C01819=1221.281,-16.840,-40.871,-179.722,5.391,148.856
C01820=1221.286,-17.090,-40.856,-179.724,5.391,148.857
C01821=1221.291,-17.339,-40.844,-179.727,5.391,148.857
C01822=1221.296,-17.589,-40.830,-179.729,5.390,148.858
C01823=1221.302,-17.838,-40.816,-179.732,5.390,148.859
C01824=1221.306,-18.088,-40.803,-179.734,5.390,148.859
C01825=1221.312,-18.337,-40.789,-179.737,5.390,148.860
C01826=1221.316,-18.587,-40.776,-179.739,5.389,148.861
C01827=1221.321,-18.837,-40.762,-179.741,5.389,148.861
C01828=1221.327,-19.086,-40.748,-179.744,5.389,148.862
C01829=1221.331,-19.336,-40.735,-179.747,5.388,148.863
C01830=1221.337,-19.585,-40.721,-179.749,5.389,148.863
C01831=1221.342,-19.835,-40.707,-179.752,5.388,148.864
C01832=1221.347,-20.084,-40.695,-179.754,5.388,148.865
C01833=1221.352,-20.334,-40.680,-179.756,5.388,148.866
C01834=1221.357,-20.583,-40.668,-179.759,5.388,148.866
C01835=1221.362,-20.833,-40.653,-179.762,5.387,148.867
C01836=1221.367,-21.082,-40.641,-179.764,5.387,148.868
C01837=1221.373,-21.333,-40.627,-179.766,5.387,148.868
C01838=1221.378,-21.582,-40.613,-179.769,5.386,148.869
C01839=1221.383,-21.832,-40.600,-179.772,5.386,148.870
C01840=1221.388,-22.081,-40.586,-179.774,5.386,148.870
C01841=1221.393,-22.350,-40.573,-179.776,5.386,148.871
C01842=1221.399,-22.620,-40.558,-179.779,5.385,148.872
C01843=1221.404,-22.889,-40.543,-179.782,5.385,148.873
C01844=1221.410,-23.158,-40.530,-179.784,5.384,148.873
C01845=1221.415,-23.408,-40.515,-179.786,5.384,148.874
C01846=1221.420,-23.657,-40.503,-179.789,5.384,148.875
C01847=1221.425,-23.908,-40.489,-179.792,5.383,148.875
C01848=1221.430,-24.156,-40.476,-179.794,5.384,148.876
C01849=1221.435,-24.407,-40.462,-179.797,5.383,148.877
C01850=1221.440,-24.656,-40.450,-179.799,5.383,148.877
C01851=1221.445,-24.906,-40.435,-179.801,5.383,148.878
C01852=1221.450,-25.155,-40.423,-179.804,5.383,148.879
C01853=1221.456,-25.405,-40.409,-179.807,5.382,148.879
C01854=1221.461,-25.654,-40.396,-179.809,5.382,148.880
C01855=1221.466,-25.904,-40.382,-179.811,5.382,148.881
C01856=1221.471,-26.154,-40.370,-179.814,5.381,148.882
C01857=1221.476,-26.403,-40.355,-179.816,5.382,148.882
C01858=1221.481,-26.653,-40.343,-179.819,5.381,148.883
C01859=1221.486,-26.903,-40.329,-179.821,5.381,148.884
C01860=1221.491,-27.152,-40.316,-179.823,5.381,148.884
C01861=1221.496,-27.401,-40.303,-179.826,5.381,148.885
C01862=1221.501,-27.651,-40.290,-179.829,5.380,148.886
C01863=1221.507,-27.901,-40.277,-179.831,5.380,148.886
C01864=1221.512,-28.150,-40.263,-179.834,5.380,148.887
C01865=1221.517,-28.400,-40.250,-179.836,5.379,148.888
C01866=1221.521,-28.650,-40.237,-179.838,5.380,148.889
C01867=1221.527,-28.899,-40.224,-179.841,5.379,148.889
C01868=1221.532,-29.149,-40.211,-179.844,5.379,148.890
C01869=1221.537,-29.398,-40.197,-179.846,5.379,148.891
C01870=1221.542,-29.648,-40.185,-179.848,5.379,148.891
C01871=1221.547,-29.898,-40.172,-179.851,5.378,148.892
C01872=1221.553,-30.147,-40.158,-179.853,5.378,148.893
C01873=1221.557,-30.397,-40.146,-179.856,5.378,148.893
C01874=1221.562,-30.646,-40.132,-179.858,5.377,148.894
C01875=1221.568,-30.896,-40.119,-179.860,5.378,148.895
C01876=1221.572,-31.146,-40.106,-179.863,5.377,148.896
C01877=1221.578,-31.395,-40.093,-179.866,5.377,148.896
C01878=1221.583,-31.645,-40.080,-179.868,5.377,148.897
C01879=1221.588,-31.895,-40.067,-179.871,5.377,148.898
C01880=1221.594,-32.144,-40.054,-179.873,5.376,148.898
C01881=1221.598,-32.394,-40.041,-179.875,5.376,148.899
C01882=1221.603,-32.643,-40.028,-179.878,5.376,148.900
C01883=1221.608,-32.892,-40.015,-179.881,5.375,148.900
C01884=1221.613,-33.143,-40.002,-179.883,5.376,148.901
C01885=1221.619,-33.392,-39.989,-179.885,5.375,148.902
C01886=1221.624,-33.641,-39.976,-179.888,5.375,148.903
C01887=1221.629,-33.892,-39.963,-179.890,5.375,148.903
C01888=1221.634,-34.141,-39.950,-179.893,5.375,148.904
C01889=1221.639,-34.390,-39.938,-179.895,5.375,148.905
C01890=1221.644,-34.641,-39.924,-179.897,5.374,148.905
C01891=1221.650,-34.890,-39.912,-179.900,5.374,148.906
C01892=1221.655,-35.139,-39.899,-179.902,5.374,148.907
C01893=1221.659,-35.389,-39.886,-179.905,5.374,148.907
C01894=1221.665,-35.639,-39.873,-179.908,5.373,148.908
C01895=1221.670,-35.888,-39.860,-179.910,5.374,148.909
C01896=1221.675,-36.138,-39.847,-179.912,5.373,148.910
C01897=1221.680,-36.388,-39.835,-179.915,5.373,148.910
C01898=1221.686,-36.637,-39.821,-179.917,5.373,148.911
C01899=1221.690,-36.887,-39.808,-179.920,5.373,148.912
C01900=1221.695,-37.137,-39.796,-179.922,5.372,148.912
C01901=1221.700,-37.386,-39.783,-179.924,5.372,148.913
C01902=1221.705,-37.636,-39.770,-179.927,5.372,148.913
C01903=1221.711,-37.886,-39.757,-179.929,5.372,148.914
C01904=1221.716,-38.135,-39.744,-179.931,5.371,148.915
C01905=1221.721,-38.384,-39.732,-179.934,5.371,148.916
C01906=1221.726,-38.634,-39.719,-179.936,5.371,148.916
C01907=1221.731,-38.883,-39.706,-179.939,5.371,148.917
C01908=1221.737,-39.133,-39.693,-179.941,5.370,148.918
C01909=1221.741,-39.383,-39.680,-179.944,5.371,148.918
C01910=1221.746,-39.632,-39.668,-179.946,5.370,148.919
C01911=1221.752,-39.882,-39.656,-179.949,5.370,148.920
C01912=1221.757,-40.132,-39.643,-179.951,5.370,148.920
C01913=1221.761,-40.382,-39.630,-179.954,5.369,148.921
C01914=1221.767,-40.631,-39.617,-179.956,5.370,148.922
C01915=1221.772,-40.881,-39.604,-179.958,5.369,148.923
C01916=1221.777,-41.130,-39.592,-179.961,5.369,148.923
C01917=1221.782,-41.380,-39.579,-179.963,5.369,148.924
C01918=1221.787,-41.630,-39.567,-179.966,5.369,148.925
C01919=1221.793,-41.879,-39.554,-179.968,5.368,148.925
C01920=1221.798,-42.129,-39.542,-179.971,5.368,148.926
C01921=1221.803,-42.379,-39.528,-179.973,5.368,148.927
C01922=1221.808,-42.628,-39.515,-179.975,5.368,148.927
C01923=1221.813,-42.878,-39.503,-179.978,5.368,148.928
C01924=1221.819,-43.127,-39.491,-179.981,5.367,148.929
C01925=1221.823,-43.378,-39.478,-179.983,5.368,148.930
C01926=1221.828,-43.627,-39.465,-179.985,5.367,148.930
C01927=1221.833,-43.876,-39.453,-179.988,5.367,148.931
C01928=1221.839,-44.125,-39.440,-179.990,5.367,148.932
C01929=1221.844,-44.375,-39.428,-179.993,5.367,148.932
C01930=1221.848,-44.625,-39.415,-179.995,5.367,148.933
C01931=1221.854,-44.875,-39.403,-179.998,5.366,148.934
C01932=1221.859,-45.124,-39.390,180.000,5.366,148.935
C01933=1221.864,-45.374,-39.378,179.998,5.366,148.935
C01934=1221.870,-45.624,-39.365,179.995,5.366,148.936
C01935=1221.875,-45.874,-39.352,179.993,5.366,148.937
C01936=1221.880,-46.124,-39.340,179.990,5.366,148.937
C01937=1221.885,-46.373,-39.328,179.988,5.365,148.938
C01938=1221.890,-46.622,-39.315,179.986,5.366,148.939
C01939=1221.896,-46.872,-39.303,179.983,5.365,148.939
C01940=1221.901,-47.121,-39.291,179.981,5.365,148.940
C01941=1221.905,-47.371,-39.278,179.978,5.365,148.941
C01942=1221.911,-47.621,-39.266,179.975,5.364,148.942
C01943=1221.916,-47.871,-39.253,179.973,5.365,148.942
C01944=1221.921,-48.120,-39.240,179.971,5.364,148.943
C01945=1221.926,-48.390,-39.228,179.968,5.364,148.944
C01946=1221.932,-48.659,-39.214,179.966,5.364,148.944
C01947=1221.938,-48.930,-39.201,179.963,5.364,148.945
C01948=1221.943,-49.200,-39.187,179.960,5.364,148.946
C01949=1221.948,-49.449,-39.174,179.958,5.364,148.947
C01950=1221.953,-49.699,-39.162,179.956,5.363,148.947
C01951=1221.959,-49.948,-39.150,179.953,5.363,148.948
C01952=1221.964,-50.198,-39.138,179.951,5.363,148.949
C01953=1221.969,-50.448,-39.125,179.948,5.362,148.949
C01954=1221.974,-50.697,-39.113,179.946,5.363,148.950
C01955=1221.978,-50.947,-39.101,179.944,5.362,148.951
C01956=1221.983,-51.197,-39.089,179.941,5.362,148.951
C01957=1221.989,-51.447,-39.077,179.939,5.362,148.952
C01958=1221.994,-51.696,-39.064,179.936,5.362,148.953
C01959=1221.999,-51.946,-39.052,179.934,5.362,148.953
C01960=1222.005,-52.195,-39.040,179.932,5.362,148.954
C01961=1222.010,-52.445,-39.028,179.929,5.361,148.955
C01962=1222.015,-52.694,-39.015,179.927,5.361,148.956
C01963=1222.021,-52.944,-39.003,179.924,5.361,148.956
C01964=1222.026,-53.194,-38.991,179.922,5.361,148.957
C01965=1222.030,-53.444,-38.979,179.919,5.361,148.958
C01966=1222.035,-53.693,-38.966,179.917,5.360,148.958
C01967=1222.040,-53.943,-38.954,179.915,5.361,148.959
C01968=1222.045,-54.193,-38.942,179.912,5.360,148.960
C01969=1222.051,-54.442,-38.930,179.910,5.361,148.961
C01970=1222.056,-54.692,-38.917,179.907,5.360,148.961
C01971=1222.061,-54.942,-38.905,179.905,5.360,148.962
C01972=1222.066,-55.191,-38.893,179.902,5.360,148.963
C01973=1222.071,-55.441,-38.882,179.900,5.359,148.963
C01974=1222.076,-55.690,-38.869,179.898,5.360,148.964
C01975=1222.082,-55.940,-38.857,179.895,5.359,148.965
C01976=1222.087,-56.190,-38.845,179.893,5.360,148.965
C01977=1222.092,-56.439,-38.833,179.890,5.359,148.966
C01978=1222.097,-56.689,-38.821,179.888,5.359,148.967
C01979=1222.102,-56.938,-38.809,179.886,5.359,148.968
C01980=1222.108,-57.188,-38.797,179.883,5.359,148.968
C01981=1222.113,-57.438,-38.785,179.881,5.359,148.969
C01982=1222.117,-57.687,-38.773,179.878,5.358,148.970
C01983=1222.122,-57.938,-38.761,179.876,5.359,148.970
C01984=1222.127,-58.187,-38.748,179.873,5.358,148.971
C01985=1222.133,-58.437,-38.736,179.871,5.358,148.972
C01986=1222.138,-58.687,-38.724,179.869,5.358,148.972
C01987=1222.143,-58.936,-38.712,179.866,5.358,148.973
C01988=1222.148,-59.186,-38.700,179.864,5.358,148.974
C01989=1222.153,-59.436,-38.689,179.862,5.357,148.974
C01990=1222.159,-59.685,-38.676,179.859,5.357,148.975
C01991=1222.163,-59.935,-38.665,179.857,5.357,148.976
C01992=1222.169,-60.185,-38.653,179.854,5.357,148.976
C01993=1222.174,-60.435,-38.641,179.852,5.357,148.977
C01994=1222.179,-60.684,-38.628,179.850,5.356,148.978
C01995=1222.184,-60.933,-38.617,179.847,5.357,148.979
C01996=1222.190,-61.183,-38.605,179.845,5.356,148.979
C01997=1222.195,-61.432,-38.593,179.842,5.356,148.980
C01998=1222.200,-61.682,-38.582,179.840,5.356,148.981
C01999=1222.205,-61.932,-38.570,179.837,5.356,148.981
C02000=1222.211,-62.181,-38.558,179.835,5.356,148.982
C02001=1222.215,-62.430,-38.546,179.833,5.356,148.983
C02002=1222.220,-62.680,-38.534,179.831,5.356,148.984
C02003=1222.226,-62.930,-38.522,179.828,5.356,148.984
C02004=1222.231,-63.180,-38.510,179.825,5.355,148.985
C02005=1222.236,-63.430,-38.499,179.823,5.355,148.986
C02006=1222.241,-63.679,-38.486,179.820,5.355,148.986
C02007=1222.247,-63.929,-38.474,179.818,5.355,148.987
C02008=1222.251,-64.179,-38.463,179.816,5.355,148.988
C02009=1222.257,-64.429,-38.451,179.814,5.355,148.988
C02010=1222.261,-64.678,-38.440,179.811,5.355,148.989
C02011=1222.267,-64.928,-38.427,179.809,5.355,148.990
C02012=1222.272,-65.178,-38.415,179.806,5.355,148.991
C02013=1222.277,-65.427,-38.404,179.803,5.354,148.991
C02014=1222.283,-65.676,-38.393,179.801,5.354,148.992
C02015=1222.288,-65.926,-38.381,179.799,5.354,148.993
C02016=1222.293,-66.176,-38.369,179.797,5.354,148.993
C02017=1222.298,-66.426,-38.358,179.794,5.354,148.994
C02018=1222.303,-66.675,-38.345,179.792,5.354,148.995
C02019=1222.308,-66.925,-38.334,179.790,5.353,148.995
C02020=1222.313,-67.175,-38.322,179.788,5.354,148.996
C02021=1222.318,-67.425,-38.310,179.785,5.353,148.997
C02022=1222.324,-67.674,-38.299,179.782,5.353,148.997
C02023=1222.329,-67.924,-38.287,179.780,5.353,148.998
C02024=1222.334,-68.173,-38.276,179.778,5.353,148.999
C02025=1222.340,-68.423,-38.264,179.775,5.353,149.000
C02026=1222.344,-68.673,-38.253,179.773,5.353,149.000
C02027=1222.350,-68.923,-38.241,179.771,5.353,149.001
C02028=1222.355,-69.172,-38.229,179.768,5.352,149.002
C02029=1222.360,-69.422,-38.218,179.766,5.353,149.002
C02030=1222.365,-69.672,-38.206,179.763,5.352,149.003
C02031=1222.371,-69.921,-38.195,179.761,5.352,149.004
C02032=1222.376,-70.171,-38.183,179.758,5.352,149.005
C02033=1222.381,-70.421,-38.172,179.756,5.352,149.005
C02034=1222.386,-70.671,-38.160,179.754,5.352,149.006
C02035=1222.391,-70.920,-38.148,179.751,5.352,149.007
C02036=1222.396,-71.170,-38.136,179.749,5.352,149.007
C02037=1222.401,-71.420,-38.125,179.746,5.352,149.008
C02038=1222.407,-71.669,-38.114,179.744,5.352,149.009
C02039=1222.412,-71.919,-38.102,179.742,5.351,149.009
C02040=1222.417,-72.169,-38.091,179.739,5.352,149.010
C02041=1222.422,-72.418,-38.079,179.737,5.351,149.011
C02042=1222.427,-72.668,-38.067,179.735,5.351,149.011
C02043=1222.433,-72.917,-38.056,179.733,5.351,149.012
C02044=1222.438,-73.167,-38.045,179.730,5.350,149.013
C02045=1222.443,-73.417,-38.033,179.728,5.351,149.013
C02046=1222.448,-73.667,-38.021,179.725,5.350,149.014
C02047=1222.453,-73.916,-38.010,179.723,5.351,149.015
C02048=1222.459,-74.166,-37.999,179.720,5.350,149.016
C02049=1222.465,-74.437,-37.986,179.718,5.351,149.016
C02050=1222.469,-74.707,-37.974,179.715,5.350,149.017
C02051=1222.475,-74.977,-37.962,179.712,5.350,149.018
C02052=1222.481,-75.248,-37.950,179.710,5.350,149.019
C02053=1222.486,-75.498,-37.938,179.708,5.350,149.019
C02054=1222.492,-75.747,-37.927,179.706,5.350,149.020
C02055=1222.496,-75.996,-37.916,179.703,5.350,149.021
C02056=1222.502,-76.246,-37.904,179.700,5.349,149.022
C02057=1222.506,-76.496,-37.893,179.698,5.350,149.022
C02058=1222.512,-76.746,-37.881,179.695,5.349,149.023
C02059=1222.518,-76.995,-37.870,179.693,5.350,149.024
C02060=1222.523,-77.245,-37.859,179.691,5.349,149.024
C02061=1222.528,-77.495,-37.847,179.689,5.349,149.025
C02062=1222.532,-77.745,-37.836,179.686,5.349,149.026
C02063=1222.538,-77.994,-37.824,179.684,5.349,149.026
C02064=1222.543,-78.244,-37.814,179.682,5.349,149.027
C02065=1222.548,-78.494,-37.803,179.680,5.349,149.028
C02066=1222.553,-78.744,-37.791,179.677,5.349,149.028
C02067=1222.559,-78.993,-37.780,179.675,5.349,149.029
C02068=1222.564,-79.243,-37.769,179.672,5.348,149.030
C02069=1222.569,-79.493,-37.757,179.670,5.349,149.030
C02070=1222.574,-79.742,-37.746,179.667,5.348,149.031
C02071=1222.580,-79.992,-37.734,179.665,5.348,149.032
C02072=1222.585,-80.242,-37.724,179.663,5.348,149.033
C02073=1222.590,-80.491,-37.713,179.660,5.348,149.033
C02074=1222.596,-80.741,-37.701,179.658,5.348,149.034
C02075=1222.600,-80.990,-37.690,179.655,5.348,149.035
C02076=1222.605,-81.241,-37.679,179.654,5.348,149.035
C02077=1222.611,-81.490,-37.668,179.651,5.347,149.036
C02078=1222.616,-81.739,-37.656,179.649,5.348,149.037
C02079=1222.621,-81.990,-37.646,179.646,5.347,149.037
C02080=1222.626,-82.239,-37.635,179.644,5.347,149.038
C02081=1222.632,-82.488,-37.623,179.641,5.347,149.039
C02082=1222.637,-82.739,-37.612,179.639,5.347,149.039
C02083=1222.641,-82.988,-37.601,179.637,5.347,149.040
C02084=1222.647,-83.238,-37.590,179.635,5.347,149.041
C02085=1222.652,-83.488,-37.579,179.632,5.347,149.042
C02086=1222.657,-83.737,-37.568,179.630,5.347,149.042
C02087=1222.662,-83.986,-37.557,179.627,5.347,149.043
C02088=1222.668,-84.237,-37.546,179.625,5.347,149.044
C02089=1222.673,-84.487,-37.534,179.622,5.347,149.044
C02090=1222.678,-84.735,-37.523,179.620,5.347,149.045
C02091=1222.683,-84.986,-37.513,179.618,5.346,149.046
C02092=1222.689,-85.236,-37.501,179.616,5.347,149.046
C02093=1222.694,-85.485,-37.491,179.613,5.346,149.047
C02094=1222.699,-85.735,-37.480,179.611,5.346,149.048
C02095=1222.704,-85.984,-37.468,179.609,5.346,149.048
C02096=1222.709,-86.234,-37.458,179.606,5.346,149.049
C02097=1222.715,-86.484,-37.446,179.604,5.346,149.050
C02098=1222.720,-86.733,-37.436,179.602,5.346,149.051
C02099=1222.725,-86.983,-37.425,179.599,5.346,149.051
C02100=1222.730,-87.233,-37.414,179.596,5.345,149.052
C02101=1222.735,-87.482,-37.403,179.594,5.346,149.053
C02102=1222.741,-87.733,-37.392,179.592,5.345,149.053
C02103=1222.746,-87.982,-37.381,179.589,5.346,149.054
C02104=1222.751,-88.232,-37.370,179.587,5.345,149.055
C02105=1222.756,-88.482,-37.359,179.585,5.345,149.055
C02106=1222.762,-88.731,-37.349,179.583,5.345,149.056
C02107=1222.766,-88.981,-37.338,179.580,5.345,149.057
C02108=1222.772,-89.231,-37.327,179.578,5.345,149.058
C02109=1222.777,-89.480,-37.316,179.576,5.345,149.058
C02110=1222.782,-89.731,-37.305,179.573,5.345,149.059
C02111=1222.788,-89.979,-37.294,179.571,5.345,149.060
C02112=1222.793,-90.230,-37.284,179.568,5.345,149.060
C02113=1222.797,-90.479,-37.272,179.566,5.345,149.061
C02114=1222.803,-90.729,-37.262,179.563,5.344,149.062
C02115=1222.808,-90.979,-37.250,179.561,5.345,149.062
C02116=1222.814,-91.228,-37.240,179.559,5.344,149.063
C02117=1222.819,-91.478,-37.229,179.557,5.344,149.064
C02118=1222.824,-91.728,-37.218,179.554,5.344,149.064
C02119=1222.829,-91.978,-37.208,179.552,5.344,149.065
C02120=1222.834,-92.227,-37.197,179.550,5.344,149.066
C02121=1222.839,-92.477,-37.186,179.548,5.344,149.067
C02122=1222.844,-92.727,-37.175,179.545,5.344,149.067
C02123=1222.850,-92.976,-37.165,179.543,5.344,149.068
C02124=1222.855,-93.226,-37.154,179.540,5.344,149.069
C02125=1222.860,-93.475,-37.143,179.538,5.344,149.069
C02126=1222.866,-93.726,-37.132,179.536,5.343,149.070
C02127=1222.871,-93.975,-37.122,179.534,5.344,149.071
C02128=1222.876,-94.225,-37.111,179.531,5.343,149.071
C02129=1222.882,-94.475,-37.100,179.529,5.343,149.072
C02130=1222.887,-94.725,-37.090,179.526,5.343,149.073
C02131=1222.892,-94.974,-37.079,179.524,5.343,149.073
C02132=1222.897,-95.224,-37.068,179.522,5.343,149.074
C02133=1222.903,-95.473,-37.058,179.519,5.343,149.075
C02134=1222.907,-95.723,-37.047,179.517,5.343,149.076
C02135=1222.913,-95.973,-37.037,179.515,5.343,149.076
C02136=1222.918,-96.223,-37.026,179.512,5.343,149.077
C02137=1222.923,-96.472,-37.015,179.510,5.343,149.077
C02138=1222.928,-96.722,-37.005,179.508,5.342,149.078
C02139=1222.934,-96.972,-36.994,179.506,5.343,149.079
C02140=1222.939,-97.222,-36.984,179.503,5.342,149.080
C02141=1222.944,-97.471,-36.973,179.501,5.343,149.080
C02142=1222.949,-97.721,-36.962,179.498,5.342,149.081
C02143=1222.955,-97.971,-36.952,179.496,5.343,149.082
C02144=1222.960,-98.221,-36.942,179.494,5.343,149.082
C02145=1222.965,-98.470,-36.931,179.491,5.343,149.083
C02146=1222.970,-98.720,-36.920,179.490,5.343,149.084
C02147=1222.975,-98.970,-36.910,179.487,5.342,149.084
C02148=1222.980,-99.220,-36.899,179.485,5.342,149.085
C02149=1222.986,-99.469,-36.888,179.482,5.342,149.086
C02150=1222.991,-99.719,-36.878,179.480,5.342,149.086
C02151=1222.996,-99.968,-36.868,179.478,5.342,149.087
C02152=1223.001,-100.219,-36.857,179.475,5.342,149.088
C02153=1223.007,-100.489,-36.846,179.473,5.342,149.089
C02154=1223.013,-100.760,-36.834,179.470,5.341,149.089
C02155=1223.018,-101.032,-36.823,179.468,5.342,149.090
C02156=1223.024,-101.303,-36.812,179.465,5.341,149.091
C02157=1223.029,-101.553,-36.801,179.463,5.342,149.091
C02158=1223.035,-101.802,-36.791,179.461,5.341,149.092
C02159=1223.039,-102.052,-36.781,179.459,5.342,149.093
C02160=1223.045,-102.301,-36.770,179.456,5.341,149.094
C02161=1223.050,-102.551,-36.760,179.454,5.342,149.094
C02162=1223.055,-102.801,-36.750,179.451,5.341,149.095
C02163=1223.061,-103.050,-36.739,179.449,5.341,149.096
C02164=1223.066,-103.301,-36.729,179.447,5.341,149.096
C02165=1223.071,-103.550,-36.719,179.445,5.341,149.097
C02166=1223.076,-103.800,-36.707,179.442,5.341,149.098
C02167=1223.081,-104.049,-36.698,179.440,5.341,149.098
C02168=1223.087,-104.299,-36.687,179.437,5.341,149.099
C02169=1223.092,-104.549,-36.677,179.435,5.341,149.100
C02170=1223.097,-104.798,-36.667,179.432,5.341,149.101
C02171=1223.102,-105.049,-36.656,179.431,5.341,149.101
C02172=1223.108,-105.298,-36.646,179.428,5.340,149.102
C02173=1223.113,-105.548,-36.636,179.426,5.341,149.102
C02174=1223.118,-105.798,-36.626,179.424,5.341,149.103
C02175=1223.123,-106.047,-36.616,179.421,5.340,149.104
C02176=1223.129,-106.297,-36.605,179.419,5.341,149.105
C02177=1223.134,-106.547,-36.595,179.417,5.340,149.105
C02178=1223.139,-106.797,-36.585,179.414,5.341,149.106
C02179=1223.144,-107.047,-36.575,179.412,5.340,149.107
C02180=1223.149,-107.296,-36.564,179.410,5.340,149.107
C02181=1223.155,-107.546,-36.554,179.408,5.340,149.108
C02182=1223.160,-107.796,-36.544,179.405,5.340,149.109
C02183=1223.165,-108.045,-36.533,179.403,5.340,149.109
C02184=1223.170,-108.295,-36.524,179.401,5.340,149.110
C02185=1223.175,-108.545,-36.513,179.398,5.340,149.111
C02186=1223.181,-108.794,-36.503,179.396,5.340,149.111
C02187=1223.186,-109.044,-36.493,179.394,5.339,149.112
C02188=1223.191,-109.294,-36.483,179.392,5.340,149.113
C02189=1223.196,-109.543,-36.473,179.389,5.339,149.113
C02190=1223.202,-109.793,-36.462,179.387,5.340,149.114
C02191=1223.207,-110.043,-36.452,179.385,5.340,149.115
C02192=1223.213,-110.293,-36.442,179.382,5.340,149.116
C02193=1223.218,-110.543,-36.433,179.380,5.340,149.116
C02194=1223.223,-110.793,-36.422,179.378,5.339,149.117
C02195=1223.228,-111.042,-36.412,179.376,5.340,149.117
C02196=1223.233,-111.292,-36.402,179.373,5.339,149.118
C02197=1223.238,-111.542,-36.392,179.371,5.340,149.119
C02198=1223.244,-111.791,-36.381,179.368,5.339,149.120
C02199=1223.249,-112.041,-36.371,179.366,5.339,149.120
C02200=1223.254,-112.290,-36.362,179.364,5.339,149.121
C02201=1223.259,-112.540,-36.351,179.362,5.339,149.122
C02202=1223.265,-112.791,-36.342,179.359,5.339,149.122
C02203=1223.270,-113.040,-36.332,179.357,5.339,149.123
C02204=1223.275,-113.290,-36.321,179.354,5.339,149.124
C02205=1223.281,-113.540,-36.311,179.352,5.339,149.124
C02206=1223.285,-113.789,-36.302,179.351,5.339,149.125
C02207=1223.291,-114.038,-36.291,179.348,5.339,149.126
C02208=1223.296,-114.289,-36.282,179.346,5.339,149.126
C02209=1223.301,-114.539,-36.272,179.343,5.338,149.127
C02210=1223.307,-114.788,-36.262,179.341,5.339,149.128
C02211=1223.312,-115.038,-36.251,179.339,5.338,149.128
C02212=1223.317,-115.288,-36.242,179.336,5.339,149.129
C02213=1223.323,-115.538,-36.232,179.334,5.338,149.130
C02214=1223.328,-115.787,-36.222,179.332,5.338,149.130
C02215=1223.333,-116.036,-36.212,179.329,5.338,149.131
C02216=1223.338,-116.287,-36.202,179.327,5.338,149.132
C02217=1223.344,-116.537,-36.192,179.325,5.338,149.133
C02218=1223.349,-116.786,-36.183,179.323,5.338,149.133
C02219=1223.354,-117.036,-36.172,179.321,5.338,149.134
C02220=1223.359,-117.286,-36.162,179.318,5.338,149.134
C02221=1223.365,-117.536,-36.153,179.316,5.338,149.135
C02222=1223.370,-117.785,-36.143,179.314,5.338,149.136
C02223=1223.375,-118.035,-36.133,179.311,5.338,149.137
C02224=1223.381,-118.285,-36.124,179.309,5.337,149.137
C02225=1223.385,-118.535,-36.114,179.307,5.338,149.138
C02226=1223.391,-118.784,-36.103,179.304,5.337,149.139
C02227=1223.397,-119.034,-36.094,179.302,5.338,149.139
C02228=1223.402,-119.284,-36.084,179.300,5.337,149.140
C02229=1223.407,-119.534,-36.074,179.298,5.338,149.141
C02230=1223.412,-119.784,-36.065,179.295,5.337,149.141
C02231=1223.417,-120.033,-36.055,179.293,5.337,149.142
C02232=1223.422,-120.282,-36.045,179.291,5.338,149.143
C02233=1223.428,-120.533,-36.035,179.289,5.337,149.143
C02234=1223.432,-120.783,-36.025,179.286,5.338,149.144
C02235=1223.438,-121.032,-36.015,179.284,5.337,149.145
C02236=1223.444,-121.282,-36.006,179.282,5.337,149.145
C02237=1223.449,-121.531,-35.996,179.280,5.337,149.146
C02238=1223.454,-121.781,-35.986,179.277,5.337,149.147
C02239=1223.459,-122.031,-35.977,179.275,5.337,149.147
C02240=1223.464,-122.281,-35.966,179.273,5.337,149.148
C02241=1223.470,-122.531,-35.958,179.271,5.337,149.149
C02242=1223.475,-122.781,-35.947,179.268,5.337,149.149
C02243=1223.480,-123.030,-35.938,179.266,5.337,149.150
C02244=1223.486,-123.280,-35.928,179.264,5.337,149.151
C02245=1223.491,-123.529,-35.919,179.262,5.337,149.151
C02246=1223.497,-123.779,-35.909,179.259,5.336,149.152
C02247=1223.501,-124.029,-35.899,179.257,5.337,149.153
C02248=1223.507,-124.279,-35.890,179.255,5.336,149.153
C02249=1223.512,-124.529,-35.880,179.252,5.337,149.154
C02250=1223.517,-124.778,-35.871,179.250,5.336,149.155
C02251=1223.523,-125.028,-35.861,179.248,5.336,149.155
C02252=1223.528,-125.278,-35.852,179.246,5.337,149.156
C02253=1223.533,-125.527,-35.842,179.243,5.336,149.157
C02254=1223.538,-125.778,-35.833,179.241,5.337,149.157
C02255=1223.543,-126.028,-35.822,179.239,5.336,149.158
C02256=1223.549,-126.277,-35.813,179.237,5.336,149.159
C02257=1223.127,-126.288,-35.850,179.233,5.340,149.161
C02258=1223.122,-126.038,-35.859,179.235,5.339,149.160
C02259=1223.117,-125.788,-35.869,179.237,5.340,149.159
C02260=1223.112,-125.538,-35.878,179.239,5.340,149.159
C02261=1223.107,-125.289,-35.888,179.242,5.340,149.158
C02262=1223.101,-125.039,-35.897,179.244,5.340,149.157
C02263=1223.096,-124.790,-35.907,179.246,5.339,149.157
C02264=1223.090,-124.539,-35.916,179.248,5.340,149.156
C02265=1223.085,-124.290,-35.926,179.250,5.340,149.155
C02266=1223.079,-124.040,-35.936,179.253,5.340,149.155
C02267=1223.075,-123.790,-35.946,179.255,5.340,149.154
C02268=1223.069,-123.540,-35.955,179.258,5.340,149.153
C02269=1223.064,-123.291,-35.965,179.260,5.340,149.153
C02270=1223.058,-123.040,-35.974,179.262,5.341,149.152
C02271=1223.053,-122.791,-35.984,179.264,5.340,149.151
C02272=1223.048,-122.542,-35.994,179.266,5.340,149.151
C02273=1223.043,-122.292,-36.003,179.269,5.340,149.150
C02274=1223.038,-122.042,-36.013,179.271,5.340,149.149
C02275=1223.033,-121.792,-36.022,179.273,5.341,149.149
C02276=1223.027,-121.542,-36.033,179.275,5.340,149.148
C02277=1223.022,-121.293,-36.042,179.278,5.341,149.147
C02278=1223.016,-121.043,-36.052,179.280,5.340,149.147
C02279=1223.012,-120.793,-36.062,179.283,5.341,149.146
C02280=1223.006,-120.543,-36.071,179.284,5.341,149.145
C02281=1223.001,-120.293,-36.081,179.287,5.341,149.145
C02282=1222.996,-120.044,-36.091,179.289,5.341,149.144
C02283=1222.990,-119.794,-36.100,179.291,5.340,149.143
C02284=1222.985,-119.545,-36.110,179.294,5.341,149.143
C02285=1222.980,-119.294,-36.121,179.296,5.340,149.142
C02286=1222.975,-119.044,-36.129,179.298,5.341,149.141
C02287=1222.969,-118.795,-36.140,179.300,5.341,149.141
C02288=1222.964,-118.546,-36.149,179.303,5.341,149.140
C02289=1222.958,-118.296,-36.159,179.305,5.341,149.139
C02290=1222.954,-118.046,-36.169,179.308,5.341,149.138
C02291=1222.948,-117.796,-36.179,179.310,5.341,149.138
C02292=1222.943,-117.547,-36.189,179.312,5.342,149.137
C02293=1222.938,-117.297,-36.198,179.314,5.341,149.137
C02294=1222.933,-117.046,-36.209,179.316,5.341,149.136
C02295=1222.928,-116.797,-36.218,179.319,5.341,149.135
C02296=1222.922,-116.547,-36.228,179.321,5.341,149.134
C02297=1222.916,-116.297,-36.238,179.323,5.342,149.134
C02298=1222.912,-116.048,-36.248,179.325,5.341,149.133
C02299=1222.906,-115.798,-36.258,179.328,5.342,149.132
C02300=1222.900,-115.548,-36.268,179.330,5.342,149.132
C02301=1222.896,-115.299,-36.277,179.332,5.342,149.131
C02302=1222.891,-115.048,-36.288,179.335,5.342,149.130
C02303=1222.885,-114.799,-36.298,179.337,5.342,149.130
C02304=1222.880,-114.550,-36.308,179.339,5.342,149.129
C02305=1222.874,-114.299,-36.317,179.342,5.342,149.128
C02306=1222.870,-114.049,-36.327,179.344,5.342,149.128
C02307=1222.864,-113.800,-36.337,179.346,5.342,149.127
C02308=1222.859,-113.550,-36.348,179.348,5.342,149.126
C02309=1222.853,-113.301,-36.358,179.350,5.342,149.126
C02310=1222.849,-113.050,-36.367,179.353,5.343,149.125
C02311=1222.843,-112.801,-36.377,179.355,5.342,149.124
C02312=1222.837,-112.551,-36.387,179.357,5.343,149.124
C02313=1222.833,-112.302,-36.397,179.360,5.342,149.123
C02314=1222.828,-112.052,-36.408,179.362,5.343,149.122
C02315=1222.822,-111.802,-36.418,179.364,5.342,149.122
C02316=1222.817,-111.553,-36.427,179.366,5.343,149.121
C02317=1222.812,-111.302,-36.437,179.369,5.343,149.120
C02318=1222.806,-111.053,-36.448,179.371,5.343,149.120
C02319=1222.801,-110.803,-36.458,179.373,5.343,149.119
C02320=1222.796,-110.553,-36.468,179.376,5.343,149.118
C02321=1222.791,-110.304,-36.478,179.378,5.343,149.117
C02322=1222.785,-110.054,-36.488,179.380,5.343,149.117
C02323=1222.780,-109.804,-36.498,179.382,5.343,149.116
C02324=1222.775,-109.555,-36.508,179.384,5.343,149.116
C02325=1222.770,-109.305,-36.519,179.387,5.343,149.115
C02326=1222.764,-109.055,-36.529,179.389,5.343,149.114
C02327=1222.759,-108.805,-36.539,179.392,5.343,149.113
C02328=1222.754,-108.556,-36.549,179.394,5.343,149.113
C02329=1222.749,-108.306,-36.559,179.396,5.344,149.112
C02330=1222.743,-108.056,-36.569,179.398,5.343,149.111
C02331=1222.738,-107.806,-36.579,179.401,5.344,149.111
C02332=1222.734,-107.556,-36.589,179.403,5.343,149.110
C02333=1222.728,-107.307,-36.599,179.406,5.344,149.109
C02334=1222.722,-107.057,-36.610,179.408,5.343,149.109
C02335=1222.717,-106.807,-36.620,179.411,5.344,149.108
C02336=1222.712,-106.557,-36.630,179.412,5.344,149.107
C02337=1222.707,-106.308,-36.640,179.415,5.344,149.107
C02338=1222.702,-106.058,-36.651,179.417,5.344,149.106
C02339=1222.696,-105.808,-36.661,179.420,5.344,149.105
C02340=1222.691,-105.559,-36.671,179.422,5.344,149.105
C02341=1222.686,-105.309,-36.682,179.424,5.344,149.104
C02342=1222.680,-105.059,-36.692,179.426,5.344,149.103
C02343=1222.676,-104.810,-36.702,179.429,5.344,149.102
C02344=1222.671,-104.560,-36.713,179.431,5.345,149.102
C02345=1222.665,-104.310,-36.723,179.433,5.344,149.101
C02346=1222.660,-104.060,-36.733,179.435,5.345,149.101
C02347=1222.654,-103.811,-36.744,179.438,5.344,149.100
C02348=1222.649,-103.560,-36.754,179.440,5.345,149.099
C02349=1222.644,-103.311,-36.764,179.442,5.344,149.098
C02350=1222.639,-103.062,-36.774,179.445,5.345,149.098
C02351=1222.634,-102.811,-36.785,179.447,5.344,149.097
C02352=1222.628,-102.562,-36.795,179.449,5.345,149.096
C02353=1222.624,-102.312,-36.806,179.451,5.345,149.096
C02354=1222.618,-102.063,-36.816,179.454,5.345,149.095
C02355=1222.613,-101.812,-36.827,179.456,5.345,149.094
C02356=1222.607,-101.563,-36.837,179.459,5.345,149.094
C02357=1222.602,-101.313,-36.847,179.461,5.345,149.093
C02358=1222.597,-101.042,-36.858,179.464,5.345,149.092
C02359=1222.591,-100.771,-36.871,179.466,5.345,149.091
C02360=1222.585,-100.500,-36.881,179.468,5.345,149.091
C02361=1222.579,-100.229,-36.893,179.471,5.346,149.090
C02362=1222.574,-99.979,-36.903,179.473,5.345,149.089
C02363=1222.569,-99.730,-36.914,179.476,5.346,149.089
C02364=1222.564,-99.479,-36.925,179.478,5.346,149.088
C02365=1222.559,-99.230,-36.934,179.481,5.346,149.087
C02366=1222.554,-98.981,-36.945,179.483,5.346,149.086
C02367=1222.549,-98.730,-36.955,179.485,5.346,149.086
C02368=1222.543,-98.482,-36.966,179.487,5.346,149.085
C02369=1222.538,-98.231,-36.977,179.490,5.346,149.085
C02370=1222.533,-97.982,-36.987,179.492,5.346,149.084
C02371=1222.528,-97.731,-36.997,179.494,5.347,149.083
C02372=1222.522,-97.483,-37.008,179.496,5.346,149.082
C02373=1222.517,-97.232,-37.019,179.499,5.346,149.082
C02374=1222.512,-96.983,-37.029,179.501,5.346,149.081
C02375=1222.507,-96.733,-37.040,179.503,5.346,149.080
C02376=1222.501,-96.484,-37.051,179.506,5.346,149.080
C02377=1222.496,-96.233,-37.061,179.508,5.346,149.079
C02378=1222.491,-95.984,-37.071,179.510,5.347,149.078
C02379=1222.486,-95.734,-37.082,179.512,5.346,149.078
C02380=1222.481,-95.485,-37.093,179.515,5.347,149.077
C02381=1222.476,-95.234,-37.103,179.517,5.346,149.076
C02382=1222.470,-94.985,-37.114,179.520,5.347,149.076
C02383=1222.465,-94.735,-37.125,179.522,5.347,149.075
C02384=1222.459,-94.485,-37.136,179.525,5.347,149.074
C02385=1222.454,-94.235,-37.146,179.527,5.347,149.073
C02386=1222.449,-93.986,-37.157,179.529,5.347,149.073
C02387=1222.444,-93.736,-37.168,179.531,5.347,149.072
C02388=1222.438,-93.486,-37.178,179.534,5.348,149.071
C02389=1222.433,-93.237,-37.189,179.536,5.347,149.071
C02390=1222.428,-92.987,-37.200,179.538,5.348,149.070
C02391=1222.423,-92.738,-37.211,179.540,5.347,149.069
C02392=1222.418,-92.487,-37.221,179.543,5.348,149.069
C02393=1222.412,-92.238,-37.232,179.545,5.347,149.068
C02394=1222.408,-91.988,-37.243,179.548,5.348,149.067
C02395=1222.402,-91.739,-37.253,179.550,5.347,149.066
C02396=1222.398,-91.489,-37.264,179.553,5.348,149.066
C02397=1222.391,-91.239,-37.275,179.555,5.347,149.065
C02398=1222.386,-90.989,-37.286,179.557,5.348,149.065
C02399=1222.381,-90.739,-37.297,179.559,5.348,149.064
C02400=1222.376,-90.490,-37.307,179.562,5.348,149.063
C02401=1222.371,-90.240,-37.319,179.564,5.348,149.062
C02402=1222.366,-89.991,-37.329,179.566,5.348,149.062
C02403=1222.361,-89.741,-37.340,179.569,5.348,149.061
C02404=1222.355,-89.491,-37.350,179.571,5.349,149.060
C02405=1222.350,-89.241,-37.362,179.573,5.348,149.060
C02406=1222.345,-88.991,-37.373,179.576,5.349,149.059
C02407=1222.340,-88.742,-37.384,179.578,5.348,149.058
C02408=1222.335,-88.492,-37.394,179.581,5.349,149.057
C02409=1222.329,-88.243,-37.405,179.583,5.348,149.057
C02410=1222.324,-87.993,-37.416,179.585,5.349,149.056
C02411=1222.319,-87.743,-37.428,179.588,5.350,149.056
C02412=1222.313,-87.493,-37.438,179.590,5.349,149.055
C02413=1222.309,-87.244,-37.449,179.592,5.350,149.054
C02414=1222.303,-86.994,-37.459,179.595,5.349,149.053
C02415=1222.298,-86.745,-37.471,179.597,5.350,149.053
C02416=1222.293,-86.494,-37.482,179.599,5.349,149.052
C02417=1222.287,-86.245,-37.493,179.602,5.350,149.051
C02418=1222.282,-85.995,-37.503,179.604,5.349,149.051
C02419=1222.278,-85.745,-37.515,179.607,5.350,149.050
C02420=1222.272,-85.496,-37.526,179.609,5.350,149.049
C02421=1222.267,-85.246,-37.537,179.612,5.350,149.048
C02422=1222.262,-84.996,-37.548,179.613,5.350,149.048
C02423=1222.256,-84.747,-37.558,179.616,5.350,149.047
C02424=1222.252,-84.497,-37.569,179.618,5.350,149.047
C02425=1222.246,-84.247,-37.581,179.621,5.351,149.046
C02426=1222.241,-83.998,-37.592,179.623,5.350,149.045
C02427=1222.236,-83.748,-37.603,179.625,5.351,149.044
C02428=1222.231,-83.498,-37.613,179.627,5.350,149.044
C02429=1222.225,-83.248,-37.625,179.630,5.351,149.043
C02430=1222.220,-82.999,-37.636,179.632,5.350,149.042
C02431=1222.215,-82.749,-37.647,179.635,5.351,149.042
C02432=1222.210,-82.500,-37.658,179.637,5.350,149.041
C02433=1222.204,-82.250,-37.670,179.640,5.351,149.040
C02434=1222.199,-81.999,-37.680,179.642,5.351,149.039
C02435=1222.194,-81.751,-37.691,179.644,5.351,149.039
C02436=1222.189,-81.501,-37.703,179.646,5.351,149.038
C02437=1222.184,-81.250,-37.714,179.649,5.352,149.038
C02438=1222.178,-81.001,-37.724,179.651,5.351,149.037
C02439=1222.174,-80.752,-37.736,179.653,5.352,149.036
C02440=1222.168,-80.502,-37.748,179.656,5.352,149.035
C02441=1222.163,-80.252,-37.758,179.658,5.352,149.035
C02442=1222.158,-80.003,-37.769,179.661,5.352,149.034
C02443=1222.153,-79.753,-37.781,179.663,5.352,149.033
C02444=1222.148,-79.502,-37.792,179.666,5.352,149.033
C02445=1222.142,-79.254,-37.803,179.668,5.352,149.032
C02446=1222.137,-79.004,-37.814,179.670,5.352,149.031
C02447=1222.132,-78.754,-37.826,179.672,5.352,149.030
C02448=1222.127,-78.504,-37.838,179.675,5.352,149.030
C02449=1222.121,-78.255,-37.848,179.677,5.352,149.029
C02450=1222.116,-78.005,-37.859,179.680,5.353,149.028
C02451=1222.111,-77.755,-37.871,179.682,5.352,149.028
C02452=1222.106,-77.505,-37.882,179.684,5.353,149.027
C02453=1222.101,-77.256,-37.893,179.686,5.353,149.026
C02454=1222.095,-77.006,-37.904,179.689,5.353,149.026
C02455=1222.091,-76.756,-37.916,179.691,5.353,149.025
C02456=1222.085,-76.506,-37.928,179.694,5.353,149.024
C02457=1222.080,-76.257,-37.938,179.696,5.354,149.024
C02458=1222.075,-76.008,-37.950,179.698,5.353,149.023
C02459=1222.069,-75.757,-37.961,179.701,5.354,149.022
C02460=1222.065,-75.508,-37.972,179.703,5.353,149.021
C02461=1222.059,-75.258,-37.984,179.706,5.354,149.021
C02462=1222.053,-74.988,-37.997,179.708,5.354,149.020
C02463=1222.048,-74.717,-38.009,179.711,5.354,149.019
C02464=1222.042,-74.447,-38.020,179.713,5.354,149.019
C02465=1222.037,-74.177,-38.033,179.716,5.354,149.018
C02466=1222.032,-73.927,-38.045,179.719,5.354,149.017
C02467=1222.027,-73.677,-38.056,179.721,5.354,149.016
C02468=1222.021,-73.428,-38.068,179.723,5.354,149.016
C02469=1222.016,-73.178,-38.078,179.725,5.354,149.015
C02470=1222.010,-72.928,-38.090,179.728,5.355,149.014
C02471=1222.006,-72.678,-38.102,179.730,5.355,149.014
C02472=1222.000,-72.428,-38.114,179.732,5.355,149.013
C02473=1221.995,-72.179,-38.124,179.735,5.355,149.012
C02474=1221.990,-71.929,-38.136,179.737,5.355,149.012
C02475=1221.985,-71.680,-38.148,179.740,5.355,149.011
C02476=1221.979,-71.430,-38.160,179.742,5.355,149.010
C02477=1221.975,-71.180,-38.171,179.745,5.355,149.009
C02478=1221.969,-70.930,-38.183,179.747,5.355,149.009
C02479=1221.964,-70.681,-38.194,179.749,5.356,149.008
C02480=1221.959,-70.431,-38.206,179.751,5.355,149.007
C02481=1221.954,-70.182,-38.217,179.754,5.356,149.007
C02482=1221.948,-69.932,-38.229,179.757,5.356,149.006
C02483=1221.944,-69.682,-38.240,179.759,5.356,149.005
C02484=1221.938,-69.432,-38.252,179.761,5.356,149.004
C02485=1221.933,-69.183,-38.263,179.764,5.356,149.004
C02486=1221.928,-68.933,-38.275,179.766,5.356,149.003
C02487=1221.922,-68.683,-38.287,179.768,5.356,149.002
C02488=1221.918,-68.434,-38.298,179.771,5.357,149.002
C02489=1221.912,-68.184,-38.310,179.773,5.357,149.001
C02490=1221.907,-67.934,-38.321,179.775,5.357,149.000
C02491=1221.902,-67.684,-38.333,179.778,5.357,149.000
C02492=1221.898,-67.435,-38.345,179.780,5.357,148.999
C02493=1221.892,-67.186,-38.356,179.783,5.358,148.998
C02494=1221.886,-66.936,-38.368,179.785,5.357,148.998
C02495=1221.881,-66.686,-38.380,179.787,5.358,148.997
C02496=1221.876,-66.437,-38.392,179.789,5.357,148.996
C02497=1221.871,-66.187,-38.403,179.792,5.358,148.996
C02498=1221.866,-65.937,-38.415,179.794,5.357,148.995
C02499=1221.860,-65.687,-38.427,179.797,5.358,148.994
C02500=1221.856,-65.437,-38.438,179.800,5.358,148.993
C02501=1221.851,-65.188,-38.450,179.802,5.358,148.993
C02502=1221.845,-64.938,-38.462,179.804,5.358,148.992
C02503=1221.840,-64.689,-38.473,179.806,5.358,148.991
C02504=1221.834,-64.439,-38.485,179.809,5.359,148.991
C02505=1221.829,-64.189,-38.497,179.811,5.358,148.990
C02506=1221.824,-63.940,-38.508,179.814,5.359,148.989
C02507=1221.819,-63.690,-38.521,179.817,5.359,148.988
C02508=1221.814,-63.440,-38.533,179.819,5.359,148.988
C02509=1221.809,-63.191,-38.544,179.821,5.359,148.987
C02510=1221.804,-62.941,-38.556,179.823,5.359,148.986
C02511=1221.798,-62.691,-38.568,179.826,5.359,148.986
C02512=1221.794,-62.442,-38.580,179.828,5.359,148.985
C02513=1221.788,-62.192,-38.592,179.831,5.360,148.984
C02514=1221.783,-61.942,-38.604,179.832,5.360,148.984
C02515=1221.778,-61.692,-38.615,179.835,5.360,148.983
C02516=1221.773,-61.443,-38.628,179.838,5.361,148.982
C02517=1221.768,-61.193,-38.639,179.840,5.360,148.982
C02518=1221.763,-60.944,-38.651,179.842,5.361,148.981
C02519=1221.758,-60.694,-38.663,179.845,5.360,148.980
C02520=1221.753,-60.444,-38.675,179.847,5.361,148.980
C02521=1221.747,-60.194,-38.687,179.849,5.360,148.979
C02522=1221.742,-59.945,-38.698,179.852,5.361,148.978
C02523=1221.737,-59.695,-38.711,179.855,5.361,148.977
C02524=1221.732,-59.445,-38.723,179.857,5.361,148.977
C02525=1221.726,-59.196,-38.735,179.859,5.361,148.976
C02526=1221.722,-58.947,-38.747,179.861,5.361,148.975
C02527=1221.717,-58.697,-38.759,179.864,5.362,148.975
C02528=1221.711,-58.447,-38.771,179.867,5.362,148.974
C02529=1221.706,-58.197,-38.783,179.869,5.362,148.973
C02530=1221.701,-57.948,-38.794,179.872,5.362,148.972
C02531=1221.696,-57.698,-38.806,179.874,5.362,148.972
C02532=1221.691,-57.448,-38.819,179.876,5.362,148.971
C02533=1221.685,-57.199,-38.831,179.878,5.362,148.970
C02534=1221.680,-56.949,-38.843,179.881,5.362,148.970
C02535=1221.676,-56.700,-38.855,179.884,5.363,148.969
C02536=1221.670,-56.450,-38.867,179.886,5.363,148.968
C02537=1221.665,-56.200,-38.879,179.889,5.363,148.968
C02538=1221.660,-55.950,-38.891,179.891,5.363,148.967
C02539=1221.654,-55.701,-38.904,179.893,5.363,148.966
C02540=1221.650,-55.451,-38.915,179.896,5.364,148.965
C02541=1221.644,-55.202,-38.927,179.898,5.363,148.965
C02542=1221.639,-54.952,-38.939,179.901,5.364,148.964
C02543=1221.634,-54.702,-38.951,179.903,5.363,148.963
C02544=1221.629,-54.453,-38.964,179.905,5.364,148.963
C02545=1221.623,-54.203,-38.976,179.907,5.364,148.962
C02546=1221.619,-53.954,-38.988,179.910,5.364,148.961
C02547=1221.614,-53.703,-39.000,179.912,5.365,148.961
C02548=1221.609,-53.454,-39.013,179.914,5.365,148.960
C02549=1221.603,-53.204,-39.025,179.917,5.365,148.959
C02550=1221.598,-52.955,-39.037,179.919,5.365,148.959
C02551=1221.593,-52.705,-39.049,179.922,5.365,148.958
C02552=1221.588,-52.456,-39.062,179.925,5.366,148.957
C02553=1221.582,-52.206,-39.074,179.927,5.365,148.957
C02554=1221.578,-51.957,-39.086,179.929,5.366,148.956
C02555=1221.573,-51.707,-39.097,179.931,5.365,148.955
C02556=1221.567,-51.457,-39.110,179.934,5.366,148.954
C02557=1221.562,-51.207,-39.122,179.937,5.366,148.954
C02558=1221.557,-50.957,-39.135,179.939,5.366,148.953
C02559=1221.552,-50.707,-39.147,179.941,5.367,148.952
C02560=1221.547,-50.458,-39.159,179.944,5.366,148.952
C02561=1221.542,-50.209,-39.172,179.946,5.367,148.951
C02562=1221.536,-49.959,-39.184,179.949,5.367,148.950
C02563=1221.531,-49.710,-39.196,179.951,5.367,148.949
C02564=1221.526,-49.460,-39.208,179.954,5.367,148.949
C02565=1221.521,-49.210,-39.221,179.956,5.367,148.948
C02566=1221.515,-48.940,-39.234,179.958,5.367,148.947
C02567=1221.510,-48.670,-39.248,179.961,5.368,148.947
C02568=1221.505,-48.401,-39.261,179.964,5.368,148.946
C02569=1221.499,-48.131,-39.274,179.966,5.368,148.945
C02570=1221.494,-47.881,-39.287,179.969,5.368,148.944
C02571=1221.488,-47.631,-39.299,179.972,5.369,148.944
C02572=1221.483,-47.382,-39.312,179.974,5.368,148.943
C02573=1221.479,-47.132,-39.324,179.976,5.369,148.942
C02574=1221.473,-46.882,-39.336,179.978,5.368,148.942
C02575=1221.468,-46.633,-39.349,179.981,5.369,148.941
C02576=1221.463,-46.383,-39.362,179.984,5.369,148.940
C02577=1221.457,-46.133,-39.373,179.986,5.369,148.939
C02578=1221.452,-45.884,-39.386,179.989,5.370,148.939
C02579=1221.448,-45.634,-39.399,179.991,5.369,148.938
C02580=1221.443,-45.385,-39.412,179.993,5.370,148.937
C02581=1221.437,-45.135,-39.424,179.996,5.370,148.937
C02582=1221.432,-44.886,-39.436,179.998,5.370,148.936
C02583=1221.427,-44.636,-39.449,-179.999,5.370,148.935
C02584=1221.422,-44.386,-39.461,-179.997,5.371,148.935
C02585=1221.417,-44.136,-39.474,-179.995,5.371,148.934
C02586=1221.412,-43.887,-39.486,-179.992,5.371,148.933
C02587=1221.407,-43.638,-39.499,-179.990,5.371,148.933
C02588=1221.402,-43.388,-39.511,-179.988,5.371,148.932
C02589=1221.396,-43.137,-39.524,-179.985,5.372,148.931
C02590=1221.391,-42.888,-39.537,-179.983,5.372,148.931
C02591=1221.386,-42.639,-39.549,-179.980,5.372,148.930
C02592=1221.381,-42.389,-39.562,-179.978,5.372,148.929
C02593=1221.376,-42.139,-39.575,-179.975,5.372,148.928
C02594=1221.371,-41.889,-39.587,-179.973,5.373,148.928
C02595=1221.366,-41.640,-39.599,-179.971,5.372,148.927
C02596=1221.360,-41.391,-39.612,-179.968,5.373,148.926
C02597=1221.356,-41.141,-39.625,-179.965,5.373,148.926
C02598=1221.350,-40.891,-39.638,-179.963,5.373,148.925
C02599=1221.345,-40.642,-39.651,-179.961,5.374,148.924
C02600=1221.340,-40.392,-39.663,-179.959,5.373,148.924
C02601=1221.335,-40.142,-39.676,-179.956,5.374,148.923
C02602=1221.330,-39.893,-39.688,-179.953,5.374,148.922
C02603=1221.325,-39.643,-39.701,-179.951,5.374,148.921
C02604=1221.320,-39.394,-39.713,-179.948,5.374,148.921
C02605=1221.314,-39.144,-39.727,-179.946,5.375,148.920
C02606=1221.309,-38.894,-39.740,-179.944,5.374,148.919
C02607=1221.304,-38.645,-39.752,-179.941,5.375,148.919
C02608=1221.299,-38.396,-39.765,-179.938,5.375,148.918
C02609=1221.295,-38.146,-39.778,-179.936,5.375,148.917
C02610=1221.288,-37.895,-39.790,-179.934,5.376,148.917
C02611=1221.283,-37.646,-39.803,-179.932,5.375,148.916
C02612=1221.279,-37.396,-39.816,-179.929,5.376,148.915
C02613=1221.274,-37.147,-39.828,-179.926,5.376,148.914
C02614=1221.268,-36.897,-39.841,-179.924,5.376,148.914
C02615=1221.263,-36.647,-39.855,-179.922,5.376,148.913
C02616=1221.258,-36.398,-39.867,-179.919,5.377,148.912
C02617=1221.253,-36.148,-39.880,-179.917,5.377,148.912
C02618=1221.248,-35.899,-39.892,-179.914,5.377,148.911
C02619=1221.243,-35.649,-39.906,-179.911,5.378,148.910
C02620=1221.237,-35.400,-39.919,-179.909,5.377,148.910
C02621=1221.232,-35.150,-39.931,-179.907,5.378,148.909
C02622=1221.228,-34.900,-39.944,-179.904,5.378,148.908
C02623=1221.222,-34.651,-39.957,-179.902,5.378,148.907
C02624=1221.217,-34.401,-39.970,-179.899,5.378,148.907
C02625=1221.212,-34.151,-39.983,-179.897,5.378,148.906
C02626=1221.206,-33.902,-39.996,-179.895,5.379,148.905
C02627=1221.202,-33.653,-40.009,-179.892,5.379,148.905
C02628=1221.197,-33.403,-40.022,-179.890,5.379,148.904
C02629=1221.192,-33.154,-40.035,-179.887,5.379,148.903
C02630=1221.186,-32.904,-40.048,-179.884,5.380,148.903
C02631=1221.182,-32.654,-40.061,-179.882,5.379,148.902
C02632=1221.176,-32.405,-40.074,-179.880,5.380,148.901
C02633=1221.171,-32.154,-40.087,-179.878,5.381,148.901
C02634=1221.166,-31.905,-40.100,-179.875,5.380,148.900
C02635=1221.161,-31.656,-40.113,-179.873,5.381,148.899
C02636=1221.156,-31.405,-40.126,-179.870,5.381,148.899
C02637=1221.151,-31.157,-40.139,-179.868,5.381,148.898
C02638=1221.146,-30.907,-40.152,-179.865,5.382,148.897
C02639=1221.140,-30.657,-40.166,-179.863,5.382,148.896
C02640=1221.135,-30.408,-40.178,-179.861,5.382,148.896
C02641=1221.131,-30.158,-40.191,-179.858,5.382,148.895
C02642=1221.125,-29.908,-40.204,-179.855,5.383,148.894
C02643=1221.120,-29.659,-40.218,-179.853,5.382,148.894
C02644=1221.116,-29.409,-40.231,-179.851,5.383,148.893
C02645=1221.110,-29.160,-40.244,-179.848,5.383,148.892
C02646=1221.105,-28.910,-40.257,-179.846,5.383,148.892
C02647=1221.099,-28.660,-40.270,-179.843,5.384,148.891
C02648=1221.095,-28.411,-40.284,-179.841,5.384,148.890
C02649=1221.090,-28.161,-40.296,-179.838,5.384,148.889
C02650=1221.084,-27.912,-40.309,-179.836,5.384,148.889
C02651=1221.080,-27.662,-40.322,-179.833,5.385,148.888
C02652=1221.074,-27.413,-40.336,-179.831,5.384,148.887
C02653=1221.070,-27.163,-40.349,-179.828,5.385,148.887
C02654=1221.064,-26.913,-40.362,-179.826,5.385,148.886
C02655=1221.059,-26.663,-40.375,-179.824,5.385,148.885
C02656=1221.054,-26.414,-40.389,-179.821,5.386,148.885
C02657=1221.049,-26.164,-40.402,-179.818,5.386,148.884
C02658=1221.044,-25.915,-40.415,-179.816,5.386,148.883
C02659=1221.038,-25.665,-40.428,-179.814,5.386,148.883
C02660=1221.034,-25.416,-40.442,-179.811,5.387,148.882
C02661=1221.028,-25.166,-40.455,-179.809,5.386,148.881
C02662=1221.024,-24.916,-40.468,-179.806,5.387,148.880
C02663=1221.018,-24.667,-40.482,-179.804,5.387,148.880
C02664=1221.013,-24.417,-40.495,-179.801,5.387,148.879
C02665=1221.008,-24.167,-40.508,-179.799,5.388,148.878
C02666=1221.003,-23.918,-40.522,-179.796,5.388,148.878
C02667=1220.998,-23.668,-40.535,-179.794,5.388,148.877
C02668=1220.993,-23.419,-40.549,-179.791,5.388,148.876
C02669=1220.987,-23.169,-40.562,-179.789,5.389,148.876
C02670=1220.983,-22.900,-40.576,-179.786,5.389,148.875
C02671=1220.977,-22.630,-40.590,-179.784,5.389,148.874
C02672=1220.972,-22.361,-40.605,-179.781,5.389,148.873
C02673=1220.966,-22.092,-40.619,-179.778,5.390,148.873
C02674=1220.961,-21.842,-40.633,-179.776,5.390,148.872
C02675=1220.956,-21.593,-40.646,-179.773,5.390,148.871
C02676=1220.951,-21.343,-40.660,-179.771,5.390,148.870
C02677=1220.945,-21.093,-40.673,-179.769,5.391,148.870
C02678=1220.941,-20.844,-40.687,-179.766,5.392,148.869
C02679=1220.935,-20.594,-40.700,-179.764,5.391,148.869
C02680=1220.930,-20.344,-40.713,-179.761,5.392,148.868
C02681=1220.925,-20.095,-40.727,-179.759,5.392,148.867
C02682=1220.920,-19.845,-40.740,-179.756,5.392,148.867
C02683=1220.915,-19.595,-40.754,-179.754,5.392,148.866
C02684=1220.910,-19.346,-40.767,-179.751,5.393,148.865
C02685=1220.905,-19.096,-40.781,-179.749,5.393,148.864
C02686=1220.899,-18.847,-40.794,-179.746,5.393,148.864
C02687=1220.895,-18.597,-40.808,-179.744,5.394,148.863
C02688=1220.889,-18.348,-40.821,-179.741,5.394,148.862
C02689=1220.884,-18.098,-40.835,-179.739,5.394,148.862
C02690=1220.880,-17.849,-40.849,-179.736,5.394,148.861
C02691=1220.874,-17.599,-40.862,-179.734,5.395,148.860
C02692=1220.869,-17.349,-40.877,-179.732,5.395,148.860
C02693=1220.864,-17.100,-40.889,-179.729,5.395,148.859
C02694=1220.859,-16.850,-40.903,-179.726,5.396,148.858
C02695=1220.853,-16.601,-40.917,-179.724,5.395,148.857
C02696=1220.849,-16.351,-40.930,-179.722,5.396,148.857
C02697=1220.844,-16.101,-40.944,-179.719,5.396,148.856
C02698=1220.838,-15.852,-40.958,-179.716,5.397,148.855
C02699=1220.834,-15.603,-40.971,-179.714,5.396,148.855
C02700=1220.828,-15.353,-40.985,-179.712,5.397,148.854
C02701=1220.823,-15.103,-40.999,-179.709,5.397,148.853
C02702=1220.819,-14.854,-41.013,-179.707,5.397,148.853
C02703=1220.813,-14.604,-41.026,-179.704,5.398,148.852
C02704=1220.808,-14.354,-41.040,-179.701,5.398,148.851
C02705=1220.803,-14.105,-41.053,-179.699,5.399,148.851
C02706=1220.798,-13.855,-41.067,-179.697,5.398,148.850
C02707=1220.793,-13.606,-41.081,-179.694,5.399,148.849
C02708=1220.788,-13.356,-41.094,-179.691,5.399,148.848
C02709=1220.783,-13.107,-41.108,-179.689,5.399,148.848
C02710=1220.778,-12.857,-41.122,-179.687,5.400,148.847
C02711=1220.773,-12.608,-41.136,-179.684,5.400,148.846
C02712=1220.768,-12.358,-41.149,-179.681,5.401,148.846
C02713=1220.763,-12.108,-41.164,-179.679,5.400,148.845
C02714=1220.758,-11.859,-41.177,-179.677,5.401,148.845
C02715=1220.752,-11.609,-41.191,-179.674,5.402,148.844
C02716=1220.748,-11.360,-41.205,-179.672,5.401,148.843
C02717=1220.743,-11.111,-41.219,-179.670,5.402,148.842
C02718=1220.738,-10.861,-41.233,-179.667,5.402,148.842
C02719=1220.732,-10.610,-41.246,-179.664,5.403,148.841
C02720=1220.727,-10.361,-41.260,-179.662,5.403,148.840
C02721=1220.723,-10.112,-41.274,-179.660,5.403,148.840
C02722=1220.718,-9.862,-41.288,-179.657,5.404,148.839
C02723=1220.712,-9.613,-41.302,-179.654,5.404,148.838
C02724=1220.707,-9.363,-41.316,-179.652,5.404,148.838
C02725=1220.702,-9.113,-41.330,-179.650,5.404,148.837
C02726=1220.697,-8.865,-41.343,-179.647,5.405,148.836
C02727=1220.692,-8.615,-41.358,-179.644,5.405,148.836
C02728=1220.687,-8.365,-41.372,-179.642,5.405,148.835
C02729=1220.682,-8.115,-41.385,-179.640,5.405,148.834
C02730=1220.676,-7.866,-41.399,-179.637,5.406,148.833
C02731=1220.671,-7.616,-41.414,-179.635,5.406,148.833
C02732=1220.667,-7.367,-41.427,-179.632,5.406,148.832
C02733=1220.662,-7.118,-41.441,-179.630,5.407,148.831
C02734=1220.657,-6.868,-41.456,-179.627,5.407,148.831
C02735=1220.652,-6.618,-41.470,-179.625,5.407,148.830
C02736=1220.647,-6.369,-41.484,-179.622,5.407,148.829
C02737=1220.641,-6.119,-41.497,-179.620,5.408,148.829
C02738=1220.636,-5.869,-41.512,-179.617,5.408,148.828
C02739=1220.632,-5.620,-41.525,-179.615,5.408,148.827
C02740=1220.627,-5.370,-41.540,-179.612,5.409,148.827
C02741=1220.621,-5.121,-41.553,-179.609,5.409,148.826
C02742=1220.616,-4.871,-41.568,-179.607,5.410,148.825
C02743=1220.611,-4.622,-41.582,-179.605,5.410,148.825
C02744=1220.606,-4.372,-41.596,-179.603,5.410,148.824
C02745=1220.601,-4.123,-41.610,-179.600,5.411,148.823
C02746=1220.596,-3.873,-41.624,-179.597,5.411,148.823
C02747=1220.591,-3.624,-41.639,-179.595,5.411,148.822
C02748=1220.586,-3.374,-41.653,-179.593,5.411,148.821
C02749=1220.581,-3.124,-41.667,-179.590,5.412,148.821
C02750=1220.576,-2.875,-41.681,-179.587,5.412,148.820
C02751=1220.571,-2.625,-41.695,-179.585,5.412,148.819
C02752=1220.566,-2.376,-41.710,-179.583,5.413,148.819
C02753=1220.561,-2.126,-41.724,-179.580,5.413,148.818
C02754=1220.556,-1.877,-41.738,-179.577,5.414,148.817
C02755=1220.551,-1.628,-41.752,-179.575,5.413,148.816
C02756=1220.546,-1.378,-41.766,-179.572,5.414,148.816
C02757=1220.541,-1.128,-41.780,-179.570,5.414,148.815
C02758=1220.536,-0.878,-41.794,-179.567,5.415,148.814
C02759=1220.531,-0.629,-41.809,-179.565,5.416,148.814
C02760=1220.525,-0.380,-41.823,-179.562,5.415,148.813
C02761=1220.521,-0.130,-41.837,-179.560,5.416,148.812
C02762=1220.516,0.120,-41.851,-179.557,5.416,148.812
C02763=1220.510,0.369,-41.867,-179.554,5.417,148.811
C02764=1220.505,0.619,-41.881,-179.552,5.416,148.810
C02765=1220.500,0.869,-41.895,-179.550,5.417,148.810
C02766=1220.495,1.118,-41.909,-179.548,5.418,148.809
C02767=1220.490,1.367,-41.924,-179.545,5.418,148.808
C02768=1220.485,1.617,-41.938,-179.543,5.418,148.808
C02769=1220.480,1.867,-41.952,-179.540,5.419,148.807
C02770=1220.475,2.116,-41.966,-179.538,5.419,148.806
C02771=1220.470,2.365,-41.981,-179.535,5.420,148.806
C02772=1220.465,2.615,-41.996,-179.532,5.420,148.805
C02773=1220.460,2.864,-42.010,-179.530,5.420,148.804
C02774=1220.455,3.133,-42.025,-179.528,5.420,148.804
C02775=1220.449,3.402,-42.040,-179.525,5.421,148.803
C02776=1220.443,3.671,-42.057,-179.522,5.421,148.802
C02777=1220.438,3.940,-42.072,-179.519,5.422,148.801
C02778=1220.433,4.190,-42.087,-179.516,5.422,148.801
C02779=1220.428,4.440,-42.101,-179.514,5.423,148.800
C02780=1220.423,4.689,-42.115,-179.512,5.422,148.799
C02781=1220.419,4.938,-42.130,-179.509,5.423,148.799
C02782=1220.413,5.187,-42.144,-179.506,5.423,148.798
C02783=1220.407,5.438,-42.159,-179.504,5.424,148.797
C02784=1220.402,5.687,-42.173,-179.502,5.425,148.797
C02785=1220.398,5.936,-42.188,-179.500,5.424,148.796
C02786=1220.393,6.186,-42.202,-179.497,5.425,148.795
C02787=1220.388,6.436,-42.217,-179.494,5.426,148.795
C02788=1220.383,6.685,-42.232,-179.492,5.426,148.794
C02789=1220.378,6.935,-42.246,-179.489,5.427,148.793
C02790=1220.373,7.185,-42.261,-179.487,5.426,148.793
C02791=1220.368,7.434,-42.276,-179.484,5.427,148.792
C02792=1220.363,7.683,-42.290,-179.482,5.427,148.791
C02793=1220.358,7.933,-42.304,-179.479,5.428,148.791
C02794=1220.353,8.182,-42.319,-179.476,5.428,148.790
C02795=1220.348,8.432,-42.334,-179.474,5.428,148.789
C02796=1220.343,8.682,-42.349,-179.472,5.429,148.788
C02797=1220.338,8.931,-42.364,-179.469,5.429,148.788
C02798=1220.333,9.180,-42.377,-179.466,5.430,148.787
C02799=1220.328,9.430,-42.392,-179.464,5.430,148.786
C02800=1220.322,9.679,-42.407,-179.461,5.430,148.786
C02801=1220.317,9.929,-42.422,-179.459,5.431,148.785
C02802=1220.313,10.178,-42.437,-179.457,5.431,148.785
C02803=1220.308,10.428,-42.451,-179.454,5.432,148.784
C02804=1220.302,10.678,-42.466,-179.451,5.432,148.783
C02805=1220.297,10.927,-42.481,-179.449,5.432,148.783
C02806=1220.292,11.176,-42.495,-179.447,5.433,148.782
C02807=1220.288,11.426,-42.510,-179.444,5.433,148.781
C02808=1220.282,11.676,-42.525,-179.441,5.434,148.780
C02809=1220.277,11.925,-42.540,-179.439,5.434,148.780
C02810=1220.272,12.174,-42.554,-179.437,5.434,148.779
C02811=1220.267,12.424,-42.570,-179.434,5.434,148.778
C02812=1220.262,12.673,-42.584,-179.431,5.435,148.778
C02813=1220.257,12.923,-42.599,-179.429,5.435,148.777
C02814=1220.252,13.173,-42.614,-179.426,5.436,148.776
C02815=1220.247,13.422,-42.629,-179.423,5.436,148.776
C02816=1220.242,13.671,-42.643,-179.422,5.437,148.775
C02817=1220.237,13.920,-42.658,-179.419,5.437,148.775
C02818=1220.232,14.171,-42.673,-179.416,5.438,148.774
C02819=1220.228,14.420,-42.688,-179.414,5.438,148.773
C02820=1220.223,14.670,-42.703,-179.411,5.439,148.772
C02821=1220.217,14.919,-42.718,-179.409,5.438,148.772
C02822=1220.212,15.169,-42.732,-179.406,5.439,148.771
C02823=1220.207,15.419,-42.748,-179.404,5.439,148.770
C02824=1220.202,15.668,-42.763,-179.401,5.440,148.770
C02825=1220.197,15.917,-42.777,-179.399,5.440,148.769
C02826=1220.192,16.167,-42.793,-179.396,5.441,148.768
C02827=1220.187,16.416,-42.807,-179.394,5.441,148.768
C02828=1220.182,16.666,-42.822,-179.391,5.441,148.767
C02829=1220.177,16.915,-42.838,-179.389,5.442,148.766
C02830=1220.172,17.165,-42.852,-179.386,5.443,148.766
C02831=1220.167,17.414,-42.868,-179.384,5.443,148.765
C02832=1220.162,17.663,-42.883,-179.381,5.444,148.765
C02833=1220.158,17.914,-42.897,-179.379,5.443,148.764
C02834=1220.152,18.163,-42.913,-179.376,5.444,148.763
C02835=1220.148,18.412,-42.928,-179.374,5.445,148.762
C02836=1220.142,18.662,-42.943,-179.371,5.445,148.762
C02837=1220.137,18.911,-42.958,-179.368,5.446,148.761
C02838=1220.132,19.161,-42.973,-179.366,5.446,148.760
C02839=1220.127,19.410,-42.988,-179.363,5.447,148.760
C02840=1220.122,19.660,-43.003,-179.361,5.446,148.759
C02841=1220.117,19.909,-43.018,-179.358,5.447,148.758
C02842=1220.113,20.159,-43.034,-179.356,5.448,148.758
C02843=1220.107,20.409,-43.048,-179.354,5.448,148.757
C02844=1220.103,20.658,-43.063,-179.351,5.449,148.757
C02845=1220.097,20.907,-43.079,-179.348,5.449,148.756
C02846=1220.093,21.156,-43.094,-179.346,5.449,148.755
C02847=1220.087,21.406,-43.109,-179.344,5.450,148.755
C02848=1220.082,21.655,-43.124,-179.341,5.450,148.754
C02849=1220.077,21.905,-43.139,-179.338,5.451,148.753
C02850=1220.073,22.154,-43.155,-179.336,5.451,148.752
C02851=1220.067,22.404,-43.170,-179.333,5.452,148.752
C02852=1220.062,22.654,-43.185,-179.330,5.452,148.751
C02853=1220.057,22.903,-43.200,-179.328,5.452,148.750
C02854=1220.052,23.152,-43.215,-179.326,5.453,148.750
C02855=1220.047,23.401,-43.231,-179.323,5.453,148.749
C02856=1220.042,23.652,-43.247,-179.321,5.454,148.749
C02857=1220.037,23.901,-43.261,-179.318,5.455,148.748
C02858=1220.032,24.151,-43.277,-179.316,5.455,148.747
C02859=1220.027,24.400,-43.292,-179.313,5.456,148.747
C02860=1220.022,24.649,-43.307,-179.310,5.456,148.746
C02861=1220.018,24.899,-43.323,-179.308,5.456,148.745
C02862=1220.012,25.148,-43.338,-179.306,5.456,148.745
C02863=1220.007,25.398,-43.354,-179.303,5.457,148.744
C02864=1220.002,25.647,-43.369,-179.300,5.458,148.743
C02865=1219.997,25.896,-43.384,-179.298,5.458,148.743
C02866=1219.993,26.147,-43.399,-179.295,5.459,148.742
C02867=1219.987,26.396,-43.415,-179.293,5.459,148.741
C02868=1219.982,26.645,-43.430,-179.290,5.460,148.741
C02869=1219.977,26.895,-43.445,-179.288,5.460,148.740
C02870=1219.972,27.145,-43.461,-179.285,5.460,148.739
C02871=1219.968,27.394,-43.476,-179.283,5.461,148.739
C02872=1219.962,27.643,-43.492,-179.280,5.461,148.738
C02873=1219.957,27.893,-43.507,-179.277,5.462,148.737
C02874=1219.952,28.142,-43.522,-179.275,5.462,148.737
C02875=1219.948,28.392,-43.538,-179.273,5.463,148.736
C02876=1219.942,28.641,-43.554,-179.270,5.464,148.735
C02877=1219.938,28.890,-43.569,-179.268,5.464,148.735
C02878=1219.932,29.159,-43.586,-179.265,5.465,148.734
C02879=1219.926,29.427,-43.603,-179.262,5.466,148.733
C02880=1219.921,29.697,-43.620,-179.259,5.466,148.733
C02881=1219.916,29.965,-43.636,-179.256,5.466,148.732
C02882=1219.911,30.215,-43.652,-179.254,5.467,148.731
C02883=1219.906,30.464,-43.667,-179.252,5.467,148.731
C02884=1219.902,30.714,-43.682,-179.249,5.467,148.730
C02885=1219.896,30.963,-43.698,-179.247,5.468,148.729
C02886=1219.891,31.213,-43.714,-179.244,5.468,148.729
C02887=1219.886,31.461,-43.730,-179.242,5.469,148.728
C02888=1219.882,31.711,-43.745,-179.239,5.470,148.727
C02889=1219.876,31.961,-43.761,-179.236,5.470,148.727
C02890=1219.871,32.210,-43.776,-179.234,5.471,148.726
C02891=1219.866,32.460,-43.792,-179.231,5.471,148.725
C02892=1219.861,32.709,-43.807,-179.229,5.471,148.725
C02893=1219.856,32.959,-43.823,-179.227,5.472,148.724
C02894=1219.851,33.209,-43.839,-179.224,5.472,148.724
C02895=1219.846,33.457,-43.855,-179.221,5.473,148.723
C02896=1219.842,33.707,-43.870,-179.219,5.473,148.722
C02897=1219.837,33.957,-43.886,-179.216,5.474,148.721
C02898=1219.831,34.206,-43.902,-179.214,5.475,148.721
C02899=1219.826,34.455,-43.917,-179.211,5.475,148.720
C02900=1219.822,34.705,-43.933,-179.209,5.476,148.720
C02901=1219.817,34.954,-43.949,-179.206,5.477,148.719
C02902=1219.811,35.203,-43.965,-179.203,5.477,148.718
C02903=1219.807,35.454,-43.981,-179.201,5.478,148.718
C02904=1219.801,35.703,-43.996,-179.199,5.477,148.717
C02905=1219.796,35.952,-44.012,-179.196,5.478,148.716
C02906=1219.792,36.202,-44.028,-179.193,5.478,148.716
C02907=1219.787,36.451,-44.043,-179.191,5.479,148.715
C02908=1219.781,36.700,-44.059,-179.188,5.480,148.714
C02909=1219.777,36.950,-44.076,-179.186,5.480,148.714
C02910=1219.771,37.199,-44.091,-179.183,5.481,148.713
C02911=1219.767,37.449,-44.107,-179.181,5.482,148.712
C02912=1219.762,37.698,-44.124,-179.178,5.482,148.712
C02913=1219.757,37.947,-44.139,-179.175,5.483,148.711
C02914=1219.752,38.197,-44.154,-179.173,5.483,148.710
C02915=1219.747,38.446,-44.171,-179.170,5.484,148.710
C02916=1219.742,38.696,-44.187,-179.168,5.485,148.709
C02917=1219.737,38.946,-44.202,-179.166,5.484,148.709
C02918=1219.732,39.194,-44.219,-179.163,5.485,148.708
C02919=1219.727,39.444,-44.235,-179.161,5.485,148.707
C02920=1219.722,39.694,-44.250,-179.158,5.486,148.707
C02921=1219.717,39.943,-44.267,-179.155,5.487,148.706
C02922=1219.712,40.193,-44.282,-179.153,5.487,148.705
C02923=1219.707,40.442,-44.299,-179.150,5.488,148.705
C02924=1219.702,40.692,-44.315,-179.148,5.489,148.704
C02925=1219.697,40.941,-44.330,-179.145,5.489,148.704
C02926=1219.693,41.190,-44.346,-179.143,5.490,148.703
C02927=1219.687,41.440,-44.362,-179.140,5.490,148.702
C02928=1219.683,41.689,-44.379,-179.137,5.491,148.701
C02929=1219.678,41.939,-44.394,-179.135,5.491,148.701
C02930=1219.673,42.188,-44.411,-179.132,5.492,148.700
C02931=1219.668,42.437,-44.426,-179.130,5.493,148.700
C02932=1219.662,42.687,-44.442,-179.127,5.493,148.699
C02933=1219.658,42.936,-44.459,-179.125,5.494,148.698
C02934=1219.652,43.186,-44.474,-179.123,5.494,148.698
C02935=1219.648,43.435,-44.491,-179.120,5.494,148.697
C02936=1219.643,43.685,-44.507,-179.117,5.495,148.696
C02937=1219.638,43.934,-44.523,-179.115,5.495,148.696
C02938=1219.633,44.183,-44.539,-179.113,5.496,148.695
C02939=1219.628,44.433,-44.555,-179.110,5.497,148.695
C02940=1219.623,44.682,-44.571,-179.107,5.497,148.694
C02941=1219.618,44.932,-44.588,-179.105,5.498,148.693
C02942=1219.613,45.181,-44.604,-179.102,5.498,148.693
C02943=1219.608,45.431,-44.621,-179.099,5.499,148.692
C02944=1219.603,45.680,-44.637,-179.097,5.500,148.691
C02945=1219.598,45.930,-44.653,-179.095,5.500,148.691
C02946=1219.593,46.179,-44.669,-179.092,5.501,148.690
C02947=1219.588,46.429,-44.685,-179.089,5.502,148.689
C02948=1219.583,46.678,-44.701,-179.087,5.502,148.689
C02949=1219.578,46.927,-44.718,-179.084,5.503,148.688
C02950=1219.573,47.176,-44.734,-179.081,5.503,148.687
C02951=1219.569,47.426,-44.750,-179.079,5.504,148.687
C02952=1219.564,47.675,-44.767,-179.077,5.505,148.686
C02953=1219.559,47.925,-44.783,-179.074,5.505,148.686
C02954=1219.554,48.174,-44.799,-179.071,5.506,148.685
C02955=1219.548,48.423,-44.816,-179.069,5.506,148.684
C02956=1219.544,48.674,-44.832,-179.066,5.507,148.684
C02957=1219.539,48.922,-44.848,-179.064,5.508,148.683
C02958=1219.534,49.172,-44.865,-179.061,5.508,148.682
C02959=1219.529,49.421,-44.881,-179.059,5.509,148.682
C02960=1219.524,49.671,-44.897,-179.056,5.510,148.681
C02961=1219.520,49.920,-44.914,-179.053,5.510,148.680
C02962=1219.514,50.170,-44.930,-179.051,5.511,148.680
C02963=1219.509,50.419,-44.947,-179.049,5.512,148.679
C02964=1219.504,50.668,-44.963,-179.046,5.512,148.679
C02965=1219.500,50.918,-44.980,-179.043,5.513,148.678
C02966=1219.495,51.168,-44.996,-179.041,5.513,148.677
C02967=1219.490,51.417,-45.012,-179.038,5.514,148.677
C02968=1219.484,51.666,-45.029,-179.036,5.514,148.676
C02969=1219.479,51.915,-45.046,-179.034,5.514,148.676
C02970=1219.475,52.165,-45.062,-179.031,5.515,148.675
C02971=1219.470,52.415,-45.078,-179.029,5.516,148.674
C02972=1219.465,52.663,-45.095,-179.026,5.516,148.674
C02973=1219.460,52.913,-45.112,-179.023,5.517,148.673
C02974=1219.455,53.162,-45.128,-179.021,5.518,148.672
C02975=1219.450,53.412,-45.145,-179.019,5.518,148.672
C02976=1219.445,53.662,-45.161,-179.016,5.519,148.671
C02977=1219.440,53.911,-45.178,-179.013,5.519,148.670
C02978=1219.435,54.160,-45.194,-179.011,5.520,148.670
C02979=1219.431,54.410,-45.211,-179.008,5.520,148.669
C02980=1219.426,54.658,-45.227,-179.006,5.521,148.669
C02981=1219.420,54.908,-45.245,-179.003,5.522,148.668
C02982=1219.415,55.177,-45.262,-179.000,5.523,148.667
C02983=1219.410,55.445,-45.280,-178.997,5.524,148.667
C02984=1219.404,55.713,-45.298,-178.995,5.524,148.666
C02985=1219.400,55.982,-45.316,-178.992,5.525,148.665
C02986=1219.394,56.231,-45.332,-178.989,5.526,148.665
C02987=1219.389,56.481,-45.350,-178.987,5.526,148.664
C02988=1219.384,56.731,-45.366,-178.984,5.527,148.663
C02989=1219.379,56.980,-45.382,-178.982,5.527,148.663
C02990=1219.374,57.229,-45.399,-178.979,5.528,148.662
C02991=1219.370,57.479,-45.416,-178.977,5.529,148.662
C02992=1219.365,57.728,-45.433,-178.974,5.529,148.661
C02993=1219.359,57.977,-45.449,-178.972,5.530,148.660
C02994=1219.355,58.227,-45.466,-178.969,5.530,148.660
C02995=1219.350,58.476,-45.483,-178.967,5.531,148.659
C02996=1219.345,58.725,-45.500,-178.964,5.532,148.658
C02997=1219.340,58.975,-45.516,-178.961,5.532,148.658
C02998=1219.335,59.225,-45.534,-178.959,5.533,148.657
C02999=1219.330,59.474,-45.550,-178.956,5.534,148.656
C03000=1219.325,59.723,-45.567,-178.954,5.534,148.656
C03001=1219.320,59.973,-45.584,-178.951,5.536,148.655
C03002=1219.316,60.222,-45.601,-178.948,5.536,148.655
C03003=1219.310,60.471,-45.618,-178.946,5.537,148.654
C03004=1219.306,60.720,-45.635,-178.943,5.538,148.653
C03005=1219.301,60.970,-45.651,-178.941,5.539,148.653
C03006=1219.296,61.219,-45.669,-178.938,5.539,148.652
C03007=1219.291,61.468,-45.685,-178.936,5.540,148.652
C03008=1219.286,61.718,-45.702,-178.933,5.540,148.651
C03009=1219.281,61.968,-45.719,-178.930,5.541,148.650
C03010=1219.276,62.217,-45.736,-178.928,5.542,148.650
C03011=1219.271,62.466,-45.753,-178.925,5.542,148.649
C03012=1219.266,62.715,-45.771,-178.923,5.543,148.649
C03013=1219.262,62.965,-45.787,-178.920,5.543,148.648
C03014=1219.257,63.214,-45.804,-178.918,5.544,148.647
C03015=1219.252,63.464,-45.821,-178.915,5.545,148.647
C03016=1219.247,63.713,-45.837,-178.913,5.545,148.646
C03017=1219.242,63.962,-45.855,-178.910,5.546,148.645
C03018=1219.237,64.212,-45.872,-178.908,5.547,148.645
C03019=1219.232,64.461,-45.889,-178.905,5.548,148.644
C03020=1219.228,64.711,-45.906,-178.903,5.548,148.644
C03021=1219.222,64.960,-45.923,-178.900,5.549,148.643
C03022=1219.218,65.209,-45.940,-178.898,5.549,148.642
C03023=1219.212,65.459,-45.958,-178.895,5.551,148.642
C03024=1219.207,65.708,-45.975,-178.892,5.552,148.641
C03025=1219.203,65.958,-45.991,-178.890,5.552,148.641
C03026=1219.197,66.206,-46.009,-178.887,5.553,148.640
C03027=1219.193,66.456,-46.026,-178.884,5.553,148.639
C03028=1219.188,66.706,-46.043,-178.882,5.554,148.639
C03029=1219.183,66.954,-46.060,-178.880,5.555,148.638
C03030=1219.178,67.204,-46.078,-178.877,5.555,148.638
C03031=1219.174,67.454,-46.094,-178.874,5.556,148.637
C03032=1219.168,67.704,-46.112,-178.872,5.557,148.636
C03033=1219.163,67.952,-46.129,-178.869,5.557,148.636
C03034=1219.158,68.201,-46.146,-178.867,5.558,148.635
C03035=1219.153,68.451,-46.163,-178.864,5.559,148.634
C03036=1219.149,68.700,-46.181,-178.862,5.559,148.634
C03037=1219.144,68.950,-46.198,-178.859,5.560,148.633
C03038=1219.139,69.199,-46.216,-178.856,5.561,148.633
C03039=1219.134,69.449,-46.232,-178.854,5.562,148.632
C03040=1219.129,69.698,-46.249,-178.851,5.563,148.631
C03041=1219.124,69.947,-46.267,-178.849,5.564,148.631
C03042=1219.119,70.196,-46.284,-178.846,5.564,148.630
C03043=1219.114,70.446,-46.302,-178.844,5.565,148.630
C03044=1219.110,70.695,-46.319,-178.841,5.565,148.629
C03045=1219.105,70.945,-46.336,-178.839,5.566,148.629
C03046=1219.100,71.194,-46.354,-178.836,5.567,148.628
C03047=1219.095,71.443,-46.371,-178.834,5.567,148.627
C03048=1219.090,71.693,-46.389,-178.831,5.568,148.627
C03049=1219.085,71.942,-46.406,-178.828,5.570,148.626
C03050=1219.081,72.191,-46.423,-178.826,5.570,148.625
C03051=1219.075,72.440,-46.440,-178.823,5.571,148.625
C03052=1219.070,72.690,-46.458,-178.820,5.571,148.624
C03053=1219.065,72.939,-46.475,-178.818,5.572,148.624
C03054=1219.061,73.188,-46.493,-178.816,5.573,148.623
C03055=1219.056,73.438,-46.510,-178.813,5.573,148.622
C03056=1219.051,73.687,-46.528,-178.810,5.574,148.622
C03057=1219.046,73.937,-46.545,-178.808,5.575,148.621
C03058=1219.041,74.186,-46.563,-178.806,5.576,148.621
C03059=1219.036,74.436,-46.580,-178.803,5.576,148.620
C03060=1219.031,74.685,-46.598,-178.800,5.578,148.620
C03061=1219.027,74.934,-46.615,-178.798,5.578,148.619
C03062=1219.022,75.183,-46.633,-178.795,5.579,148.618
C03063=1219.017,75.433,-46.650,-178.792,5.580,148.618
C03064=1219.012,75.682,-46.668,-178.790,5.581,148.617
C03065=1219.007,75.932,-46.686,-178.788,5.581,148.616
C03066=1219.003,76.180,-46.703,-178.785,5.582,148.616
C03067=1218.997,76.430,-46.720,-178.782,5.582,148.615
C03068=1218.992,76.679,-46.738,-178.780,5.584,148.615
C03069=1218.987,76.929,-46.756,-178.777,5.585,148.614
C03070=1218.983,77.178,-46.773,-178.774,5.585,148.613
C03071=1218.978,77.427,-46.791,-178.772,5.586,148.613
C03072=1218.973,77.676,-46.809,-178.770,5.587,148.612
C03073=1218.968,77.926,-46.826,-178.767,5.587,148.612
C03074=1218.963,78.175,-46.844,-178.764,5.588,148.611
C03075=1218.958,78.425,-46.862,-178.762,5.589,148.611
C03076=1218.954,78.674,-46.879,-178.760,5.589,148.610
C03077=1218.949,78.923,-46.897,-178.756,5.591,148.609
C03078=1218.944,79.172,-46.915,-178.754,5.591,148.609
C03079=1218.939,79.422,-46.932,-178.752,5.592,148.608
C03080=1218.934,79.671,-46.950,-178.749,5.593,148.608
C03081=1218.929,79.921,-46.968,-178.746,5.594,148.607
C03082=1218.924,80.170,-46.986,-178.744,5.594,148.606
C03083=1218.919,80.420,-47.003,-178.742,5.595,148.606
C03084=1218.914,80.669,-47.021,-178.738,5.596,148.605
C03085=1218.910,80.918,-47.039,-178.736,5.597,148.605
C03086=1218.905,81.186,-47.058,-178.733,5.598,148.604
C03087=1218.899,81.455,-47.077,-178.731,5.599,148.603
C03088=1218.894,81.723,-47.096,-178.728,5.600,148.603
C03089=1218.888,81.992,-47.116,-178.725,5.601,148.602
C03090=1218.884,82.240,-47.134,-178.723,5.601,148.601
C03091=1218.879,82.490,-47.152,-178.720,5.602,148.601
C03092=1218.874,82.739,-47.169,-178.718,5.603,148.600
C03093=1218.869,82.989,-47.187,-178.715,5.604,148.600
C03094=1218.864,83.238,-47.205,-178.712,5.605,148.599
C03095=1218.859,83.487,-47.223,-178.709,5.605,148.598
C03096=1218.854,83.736,-47.241,-178.707,5.606,148.598
C03097=1218.850,83.986,-47.259,-178.705,5.607,148.597
C03098=1218.845,84.235,-47.277,-178.702,5.607,148.597
C03099=1218.840,84.484,-47.295,-178.700,5.608,148.596
C03100=1218.835,84.733,-47.313,-178.697,5.610,148.596
C03101=1218.830,84.983,-47.330,-178.694,5.610,148.595
C03102=1218.825,85.232,-47.348,-178.692,5.611,148.595
C03103=1218.820,85.482,-47.366,-178.689,5.612,148.594
C03104=1218.815,85.731,-47.384,-178.687,5.612,148.593
C03105=1218.811,85.981,-47.403,-178.685,5.613,148.593
C03106=1218.806,86.230,-47.421,-178.681,5.615,148.592
C03107=1218.801,86.479,-47.439,-178.679,5.615,148.592
C03108=1218.796,86.728,-47.457,-178.676,5.616,148.591
C03109=1218.791,86.977,-47.474,-178.674,5.617,148.590
C03110=1218.786,87.227,-47.492,-178.671,5.617,148.590
C03111=1218.781,87.476,-47.511,-178.669,5.618,148.589
C03112=1218.776,87.726,-47.529,-178.666,5.620,148.589
C03113=1218.772,87.975,-47.547,-178.663,5.620,148.588
C03114=1218.767,88.224,-47.565,-178.661,5.621,148.587
C03115=1218.762,88.473,-47.583,-178.659,5.622,148.587
C03116=1218.757,88.723,-47.601,-178.656,5.622,148.586
C03117=1218.753,88.972,-47.620,-178.653,5.624,148.586
C03118=1218.748,89.221,-47.638,-178.651,5.625,148.585
C03119=1218.743,89.470,-47.656,-178.648,5.625,148.585
C03120=1218.738,89.719,-47.674,-178.645,5.626,148.584
C03121=1218.732,89.969,-47.693,-178.643,5.627,148.584
C03122=1218.728,90.219,-47.711,-178.641,5.628,148.583
C03123=1218.723,90.468,-47.729,-178.638,5.629,148.582
C03124=1218.718,90.717,-47.747,-178.635,5.630,148.582
C03125=1218.713,90.966,-47.765,-178.633,5.631,148.581
C03126=1218.709,91.215,-47.784,-178.630,5.631,148.581
C03127=1218.704,91.465,-47.802,-178.628,5.632,148.580
C03128=1218.699,91.714,-47.821,-178.625,5.633,148.579
C03129=1218.694,91.963,-47.839,-178.622,5.634,148.579
C03130=1218.689,92.213,-47.857,-178.620,5.635,148.578
C03131=1218.685,92.462,-47.876,-178.617,5.636,148.578
C03132=1218.680,92.711,-47.894,-178.615,5.636,148.577
C03133=1218.674,92.961,-47.912,-178.612,5.638,148.577
C03134=1218.669,93.210,-47.930,-178.610,5.639,148.576
C03135=1218.665,93.460,-47.949,-178.607,5.639,148.575
C03136=1218.661,93.708,-47.967,-178.605,5.640,148.575
C03137=1218.656,93.957,-47.985,-178.602,5.641,148.574
C03138=1218.650,94.207,-48.004,-178.599,5.642,148.574
C03139=1218.646,94.457,-48.022,-178.597,5.643,148.573
C03140=1218.641,94.705,-48.041,-178.594,5.644,148.573
C03141=1218.636,94.954,-48.059,-178.592,5.644,148.572
C03142=1218.631,95.204,-48.078,-178.589,5.646,148.572
C03143=1218.627,95.453,-48.097,-178.586,5.647,148.571
C03144=1218.622,95.702,-48.115,-178.584,5.648,148.570
C03145=1218.617,95.951,-48.133,-178.582,5.648,148.570
C03146=1218.612,96.201,-48.152,-178.579,5.649,148.569
C03147=1218.607,96.450,-48.170,-178.576,5.650,148.569
C03148=1218.602,96.699,-48.188,-178.574,5.651,148.568
C03149=1218.597,96.949,-48.208,-178.571,5.652,148.567
C03150=1218.592,97.198,-48.226,-178.569,5.653,148.567
C03151=1218.588,97.447,-48.244,-178.566,5.654,148.566
C03152=1218.583,97.697,-48.263,-178.563,5.655,148.566
C03153=1218.578,97.946,-48.281,-178.561,5.656,148.565
C03154=1218.573,98.195,-48.300,-178.558,5.656,148.565
C03155=1218.568,98.445,-48.319,-178.556,5.657,148.564
C03156=1218.563,98.694,-48.337,-178.553,5.659,148.564
C03157=1218.559,98.943,-48.356,-178.550,5.659,148.563
C03158=1218.554,99.193,-48.375,-178.548,5.660,148.563
C03159=1218.549,99.441,-48.393,-178.546,5.661,148.562
C03160=1218.544,99.690,-48.411,-178.542,5.662,148.561
C03161=1218.539,99.940,-48.431,-178.540,5.663,148.561
C03162=1218.535,100.189,-48.449,-178.538,5.664,148.560
C03163=1218.529,100.438,-48.468,-178.536,5.665,148.560
C03164=1218.525,100.688,-48.487,-178.532,5.666,148.559
C03165=1218.520,100.937,-48.505,-178.530,5.667,148.559
C03166=1218.515,101.187,-48.524,-178.528,5.668,148.558
C03167=1218.511,101.435,-48.543,-178.525,5.668,148.557
C03168=1218.505,101.685,-48.562,-178.522,5.670,148.557
C03169=1218.501,101.934,-48.581,-178.520,5.671,148.556
C03170=1218.496,102.183,-48.599,-178.517,5.671,148.556
C03171=1218.491,102.433,-48.618,-178.515,5.672,148.555
C03172=1218.487,102.681,-48.637,-178.512,5.674,148.555
C03173=1218.481,102.931,-48.655,-178.509,5.674,148.554
C03174=1218.477,103.180,-48.675,-178.507,5.675,148.554
C03175=1218.471,103.430,-48.693,-178.504,5.676,148.553
C03176=1218.467,103.679,-48.712,-178.502,5.677,148.553
C03177=1218.462,103.928,-48.731,-178.499,5.678,148.552
C03178=1218.457,104.177,-48.749,-178.497,5.679,148.551
C03179=1218.452,104.426,-48.769,-178.494,5.680,148.551
C03180=1218.447,104.676,-48.787,-178.491,5.681,148.550
C03181=1218.443,104.925,-48.807,-178.489,5.682,148.550
C03182=1218.438,105.174,-48.825,-178.486,5.683,148.549
C03183=1218.433,105.424,-48.844,-178.483,5.684,148.549
C03184=1218.428,105.672,-48.863,-178.481,5.685,148.548
C03185=1218.424,105.922,-48.883,-178.479,5.686,148.548
C03186=1218.419,106.171,-48.901,-178.476,5.687,148.547
C03187=1218.414,106.421,-48.920,-178.473,5.688,148.546
C03188=1218.409,106.669,-48.939,-178.471,5.689,148.546
C03189=1218.404,106.918,-48.958,-178.469,5.690,148.545
C03190=1218.399,107.187,-48.979,-178.465,5.691,148.545
C03191=1218.393,107.455,-48.999,-178.463,5.692,148.544
C03192=1218.389,107.724,-49.020,-178.460,5.693,148.544
C03193=1218.383,107.992,-49.040,-178.457,5.694,148.543
C03194=1218.379,108.242,-49.060,-178.455,5.695,148.542
C03195=1218.374,108.490,-49.078,-178.452,5.696,148.542
C03196=1218.369,108.740,-49.098,-178.449,5.697,148.541
C03197=1218.364,108.989,-49.117,-178.447,5.698,148.541
C03198=1218.360,109.239,-49.136,-178.444,5.699,148.540
C03199=1218.354,109.488,-49.155,-178.442,5.700,148.540
C03200=1218.350,109.737,-49.174,-178.439,5.701,148.539
C03201=1218.345,109.986,-49.193,-178.437,5.701,148.539
C03202=1218.340,110.235,-49.213,-178.434,5.703,148.538
C03203=1218.336,110.485,-49.231,-178.432,5.704,148.538
C03204=1218.331,110.734,-49.251,-178.429,5.704,148.537
C03205=1218.326,110.984,-49.270,-178.426,5.706,148.537
C03206=1218.321,111.232,-49.289,-178.424,5.707,148.536
C03207=1218.316,111.482,-49.309,-178.422,5.708,148.536
C03208=1218.311,111.731,-49.328,-178.418,5.709,148.535
C03209=1218.307,111.980,-49.347,-178.416,5.710,148.534
C03210=1218.302,112.229,-49.366,-178.414,5.711,148.534
C03211=1218.297,112.478,-49.386,-178.410,5.712,148.533
C03212=1218.293,112.728,-49.405,-178.408,5.713,148.533
C03213=1218.288,112.976,-49.424,-178.406,5.714,148.532
C03214=1218.283,113.226,-49.444,-178.404,5.715,148.532
C03215=1218.277,113.475,-49.462,-178.400,5.716,148.531
C03216=1218.273,113.725,-49.481,-178.398,5.717,148.531
C03217=1218.268,113.974,-49.501,-178.396,5.718,148.530
C03218=1218.263,114.223,-49.520,-178.392,5.719,148.529
C03219=1218.258,114.473,-49.540,-178.390,5.720,148.529
C03220=1218.254,114.721,-49.559,-178.388,5.721,148.528
C03221=1218.249,114.970,-49.579,-178.385,5.723,148.528
C03222=1218.244,115.219,-49.598,-178.382,5.723,148.527
C03223=1218.239,115.469,-49.618,-178.380,5.724,148.527
C03224=1218.235,115.718,-49.637,-178.377,5.726,148.526
C03225=1218.230,115.967,-49.656,-178.375,5.727,148.526
C03226=1218.225,116.216,-49.676,-178.372,5.727,148.525
C03227=1218.220,116.466,-49.696,-178.370,5.729,148.525
C03228=1218.215,116.715,-49.715,-178.367,5.730,148.524
C03229=1218.211,116.964,-49.734,-178.364,5.730,148.524
C03230=1218.206,117.213,-49.753,-178.362,5.732,148.523
C03231=1218.201,117.462,-49.773,-178.359,5.733,148.523
C03232=1218.196,117.712,-49.793,-178.357,5.734,148.522
C03233=1218.191,117.960,-49.813,-178.354,5.735,148.522
C03234=1218.186,118.210,-49.832,-178.352,5.736,148.521
C03235=1218.182,118.459,-49.851,-178.349,5.737,148.520
C03236=1218.177,118.708,-49.871,-178.346,5.738,148.520
C03237=1218.172,118.958,-49.890,-178.344,5.739,148.519
C03238=1218.168,119.207,-49.910,-178.341,5.741,148.519
C03239=1218.163,119.455,-49.930,-178.339,5.741,148.518
C03240=1218.158,119.705,-49.950,-178.336,5.742,148.518
C03241=1218.153,119.955,-49.969,-178.333,5.744,148.517
C03242=1218.148,120.203,-49.989,-178.331,5.745,148.517
C03243=1218.143,120.452,-50.009,-178.329,5.745,148.516
C03244=1218.139,120.702,-50.028,-178.326,5.747,148.516
C03245=1218.135,120.951,-50.048,-178.323,5.748,148.515
C03246=1218.129,121.200,-50.067,-178.321,5.749,148.515
C03247=1218.125,121.449,-50.087,-178.318,5.750,148.514
C03248=1218.120,121.699,-50.107,-178.316,5.751,148.514
C03249=1218.115,121.947,-50.126,-178.313,5.753,148.513
C03250=1218.110,122.197,-50.146,-178.310,5.753,148.513
C03251=1218.106,122.446,-50.166,-178.308,5.754,148.512
C03252=1218.101,122.696,-50.186,-178.305,5.756,148.512
C03253=1218.095,122.944,-50.205,-178.303,5.756,148.511
C03254=1218.091,123.193,-50.226,-178.300,5.757,148.511
C03255=1218.086,123.443,-50.245,-178.297,5.759,148.510
C03256=1218.082,123.692,-50.265,-178.295,5.760,148.509
C03257=1218.077,123.941,-50.285,-178.292,5.761,148.509
C03258=1218.072,124.190,-50.305,-178.289,5.762,148.508
C03259=1218.067,124.439,-50.325,-178.287,5.763,148.508
C03260=1218.063,124.689,-50.345,-178.284,5.764,148.507
C03261=1218.057,124.938,-50.364,-178.282,5.765,148.507
C03262=1218.053,125.187,-50.384,-178.279,5.766,148.506
C03263=1218.048,125.436,-50.404,-178.277,5.768,148.506
C03264=1218.044,125.685,-50.424,-178.275,5.769,148.506
C03265=1218.039,125.935,-50.444,-178.272,5.770,148.505
C03266=1218.034,126.183,-50.464,-178.269,5.771,148.505
C03267=1218.029,126.432,-50.484,-178.267,5.772,148.504
C03268=1218.024,126.682,-50.503,-178.264,5.773,148.504
C03269=1218.020,126.931,-50.524,-178.261,5.774,148.503
C03270=1218.015,127.181,-50.543,-178.259,5.776,148.503
C03271=1218.010,127.429,-50.563,-178.256,5.777,148.502
C03272=1218.005,127.679,-50.584,-178.254,5.777,148.501
C03273=1218.000,127.928,-50.604,-178.251,5.779,148.501
C03274=1217.996,128.177,-50.624,-178.249,5.780,148.500
C03275=1217.991,128.426,-50.644,-178.246,5.781,148.500
C03276=1217.987,128.675,-50.664,-178.244,5.782,148.499
C03277=1217.981,128.924,-50.684,-178.241,5.783,148.499
C03278=1217.977,129.173,-50.704,-178.238,5.785,148.498
C03279=1217.972,129.423,-50.724,-178.236,5.785,148.498
C03280=1217.968,129.671,-50.744,-178.233,5.787,148.497
C03281=1217.962,129.921,-50.765,-178.230,5.788,148.497
C03282=1217.958,130.170,-50.785,-178.228,5.790,148.496
C03283=1217.953,130.419,-50.805,-178.225,5.790,148.496
C03284=1217.948,130.668,-50.824,-178.223,5.791,148.495
C03285=1217.944,130.917,-50.845,-178.220,5.793,148.495
C03286=1217.939,131.166,-50.865,-178.218,5.794,148.494
C03287=1217.934,131.416,-50.885,-178.215,5.795,148.494
C03288=1217.929,131.665,-50.906,-178.212,5.796,148.493
C03289=1217.925,131.914,-50.926,-178.210,5.797,148.493
C03290=1217.920,132.163,-50.946,-178.207,5.798,148.492
C03291=1217.915,132.413,-50.967,-178.205,5.799,148.492
C03292=1217.910,132.661,-50.987,-178.202,5.801,148.491
C03293=1217.905,132.910,-51.006,-178.200,5.802,148.491
C03294=1217.900,133.179,-51.029,-178.197,5.803,148.490
C03295=1217.895,133.448,-51.050,-178.194,5.804,148.490
C03296=1217.890,133.716,-51.073,-178.191,5.806,148.489
C03297=1217.884,133.985,-51.094,-178.188,5.807,148.489
C03298=1217.880,134.234,-51.115,-178.186,5.808,148.488
C03299=1217.875,134.483,-51.135,-178.183,5.810,148.488
C03300=1217.871,134.732,-51.155,-178.181,5.811,148.487
C03301=1217.866,134.982,-51.176,-178.178,5.812,148.487
C03302=1217.861,135.231,-51.196,-178.175,5.813,148.486
C03303=1217.857,135.480,-51.216,-178.173,5.814,148.486
C03304=1217.852,135.729,-51.237,-178.170,5.815,148.485
C03305=1217.847,135.978,-51.258,-178.168,5.816,148.485
C03306=1217.843,136.227,-51.278,-178.165,5.818,148.484
C03307=1217.837,136.476,-51.299,-178.163,5.819,148.484
C03308=1217.832,136.725,-51.318,-178.160,5.821,148.483
C03309=1217.828,136.974,-51.339,-178.157,5.821,148.483
C03310=1217.823,137.224,-51.360,-178.155,5.823,148.482
C03311=1217.818,137.472,-51.380,-178.152,5.824,148.482
C03312=1217.814,137.721,-51.401,-178.150,5.825,148.481
C03313=1217.808,137.971,-51.421,-178.147,5.826,148.481
C03314=1217.804,138.220,-51.442,-178.145,5.827,148.480
C03315=1217.800,138.469,-51.462,-178.142,5.829,148.480
C03316=1217.794,138.718,-51.483,-178.140,5.829,148.479
C03317=1217.790,138.967,-51.504,-178.137,5.831,148.479
C03318=1217.785,139.216,-51.525,-178.134,5.832,148.478
C03319=1217.780,139.466,-51.544,-178.132,5.834,148.478
C03320=1217.776,139.715,-51.565,-178.129,5.835,148.478
C03321=1217.770,139.964,-51.586,-178.126,5.836,148.477
C03322=1217.766,140.213,-51.606,-178.124,5.837,148.477
C03323=1217.761,140.462,-51.627,-178.121,5.839,148.476
C03324=1217.757,140.712,-51.648,-178.119,5.839,148.475
C03325=1217.753,140.961,-51.668,-178.116,5.841,148.475
C03326=1217.748,141.209,-51.690,-178.114,5.842,148.474
C03327=1217.743,141.458,-51.710,-178.111,5.844,148.474
C03328=1217.738,141.707,-51.731,-178.108,5.844,148.473
C03329=1217.734,141.956,-51.751,-178.106,5.846,148.473
C03330=1217.728,142.206,-51.772,-178.104,5.847,148.473
C03331=1217.724,142.455,-51.793,-178.100,5.849,148.472
C03332=1217.719,142.704,-51.814,-178.098,5.850,148.472
C03333=1217.714,142.953,-51.834,-178.095,5.851,148.471
C03334=1217.709,143.202,-51.855,-178.093,5.852,148.471
C03335=1217.705,143.451,-51.875,-178.090,5.854,148.470
C03336=1217.700,143.700,-51.896,-178.088,5.854,148.470
C03337=1217.696,143.949,-51.917,-178.085,5.856,148.469
C03338=1217.691,144.199,-51.939,-178.083,5.857,148.469
C03339=1217.686,144.448,-51.959,-178.080,5.859,148.468
C03340=1217.681,144.697,-51.980,-178.078,5.860,148.468
C03341=1217.677,144.946,-52.000,-178.075,5.861,148.467
C03342=1217.672,145.195,-52.021,-178.072,5.862,148.467
C03343=1217.667,145.444,-52.043,-178.070,5.864,148.467
C03344=1217.662,145.693,-52.063,-178.067,5.865,148.466
C03345=1217.657,145.942,-52.084,-178.065,5.866,148.466
C03346=1217.653,146.191,-52.105,-178.062,5.867,148.465
C03347=1217.649,146.440,-52.127,-178.059,5.869,148.465
C03348=1217.644,146.689,-52.147,-178.057,5.870,148.464
C03349=1217.639,146.938,-52.168,-178.054,5.871,148.464
C03350=1217.634,147.188,-52.189,-178.052,5.872,148.463
C03351=1217.630,147.436,-52.210,-178.049,5.874,148.463
C03352=1217.624,147.685,-52.231,-178.047,5.875,148.462
C03353=1217.619,147.934,-52.252,-178.044,5.876,148.462
C03354=1217.615,148.184,-52.273,-178.041,5.877,148.461
C03355=1217.611,148.433,-52.295,-178.039,5.879,148.461
C03356=1217.606,148.682,-52.315,-178.037,5.880,148.460
C03357=1217.601,148.931,-52.336,-178.033,5.881,148.460
C03358=1217.596,149.180,-52.358,-178.031,5.883,148.459
C03359=1217.592,149.429,-52.378,-178.029,5.884,148.459
C03360=1217.587,149.678,-52.400,-178.025,5.886,148.458
C03361=1217.582,149.927,-52.421,-178.023,5.887,148.458
C03362=1217.577,150.176,-52.442,-178.021,5.888,148.458
C03363=1217.573,150.425,-52.463,-178.018,5.889,148.457
C03364=1217.568,150.674,-52.484,-178.015,5.891,148.457
C03365=1217.563,150.923,-52.506,-178.013,5.892,148.456
C03366=1217.559,151.172,-52.526,-178.010,5.893,148.456
C03367=1217.554,151.422,-52.547,-178.008,5.894,148.455
C03368=1217.549,151.670,-52.569,-178.005,5.896,148.455
C03369=1217.544,151.920,-52.590,-178.002,5.897,148.454
C03370=1217.540,152.169,-52.612,-178.000,5.898,148.454
C03371=1217.535,152.418,-52.633,-177.997,5.900,148.453
C03372=1217.530,152.666,-52.654,-177.995,5.901,148.453
C03373=1217.526,152.916,-52.676,-177.992,5.903,148.452
C03374=1217.522,153.165,-52.697,-177.990,5.904,148.452
C03375=1217.516,153.414,-52.718,-177.987,5.905,148.451
C03376=1217.511,153.663,-52.739,-177.985,5.906,148.451
C03377=1217.507,153.913,-52.761,-177.982,5.908,148.451
C03378=1217.502,154.161,-52.782,-177.979,5.909,148.450
C03379=1217.498,154.410,-52.803,-177.977,5.910,148.450
C03380=1217.493,154.659,-52.824,-177.974,5.912,148.449
C03381=1217.488,154.908,-52.846,-177.972,5.913,148.449
C03382=1217.483,155.157,-52.867,-177.969,5.915,148.448
C03383=1217.478,155.406,-52.889,-177.967,5.916,148.448
C03384=1217.473,155.655,-52.910,-177.964,5.917,148.447
C03385=1217.470,155.904,-52.931,-177.961,5.919,148.447
C03386=1217.465,156.153,-52.953,-177.959,5.920,148.447
C03387=1217.460,156.402,-52.974,-177.956,5.921,148.446
C03388=1217.455,156.652,-52.996,-177.954,5.922,148.446
C03389=1217.451,156.900,-53.018,-177.951,5.924,148.445
C03390=1217.445,157.149,-53.039,-177.948,5.925,148.445
C03391=1217.441,157.399,-53.061,-177.946,5.927,148.444
C03392=1217.436,157.647,-53.083,-177.943,5.928,148.444
C03393=1217.432,157.896,-53.103,-177.941,5.929,148.443
C03394=1217.427,158.146,-53.125,-177.938,5.931,148.443
C03395=1217.423,158.394,-53.147,-177.936,5.932,148.442
C03396=1217.417,158.644,-53.168,-177.933,5.934,148.442
C03397=1217.413,158.893,-53.190,-177.930,5.935,148.442
C03398=1217.408,159.162,-53.213,-177.928,5.936,148.441
C03399=1217.403,159.431,-53.236,-177.925,5.938,148.441
C03400=1217.398,159.700,-53.260,-177.922,5.939,148.440
C03401=1217.393,159.969,-53.283,-177.919,5.941,148.440
C03402=1217.388,160.218,-53.304,-177.917,5.942,148.439
C03403=1217.383,160.466,-53.326,-177.914,5.944,148.439
C03404=1217.379,160.716,-53.348,-177.911,5.946,148.438
C03405=1217.374,160.964,-53.370,-177.909,5.946,148.438
C03406=1217.370,161.214,-53.391,-177.906,5.948,148.437
C03407=1217.365,161.463,-53.413,-177.904,5.949,148.437
C03408=1217.360,161.712,-53.434,-177.901,5.950,148.436
C03409=1217.356,161.961,-53.456,-177.898,5.952,148.436
C03410=1217.351,162.210,-53.478,-177.896,5.953,148.436
C03411=1217.346,162.459,-53.500,-177.893,5.955,148.435
C03412=1217.342,162.708,-53.522,-177.890,5.957,148.435
C03413=1217.337,162.956,-53.544,-177.888,5.958,148.434
C03414=1217.332,163.206,-53.566,-177.886,5.959,148.434
C03415=1217.327,163.455,-53.587,-177.883,5.960,148.434
C03416=1217.322,163.705,-53.609,-177.880,5.962,148.433
C03417=1217.317,163.953,-53.631,-177.878,5.964,148.433
C03418=1217.313,164.203,-53.653,-177.876,5.965,148.432
C03419=1217.308,164.451,-53.675,-177.872,5.966,148.432
C03420=1217.303,164.700,-53.696,-177.870,5.968,148.431
C03421=1217.299,164.949,-53.718,-177.868,5.969,148.431
C03422=1217.294,165.198,-53.740,-177.865,5.971,148.431
C03423=1217.290,165.447,-53.762,-177.862,5.971,148.430
C03424=1217.285,165.696,-53.784,-177.860,5.973,148.430
C03425=1217.281,165.945,-53.806,-177.857,5.975,148.429
C03426=1217.275,166.194,-53.828,-177.855,5.976,148.429
C03427=1217.271,166.443,-53.850,-177.852,5.977,148.428
C03428=1217.266,166.692,-53.872,-177.849,5.979,148.428
C03429=1217.262,166.941,-53.894,-177.847,5.980,148.427
C03430=1217.257,167.190,-53.916,-177.844,5.982,148.427
C03431=1217.253,167.439,-53.938,-177.841,5.984,148.427
C03432=1217.248,167.687,-53.960,-177.839,5.985,148.426
C03433=1217.243,167.937,-53.983,-177.837,5.986,148.426
C03434=1217.238,168.186,-54.004,-177.834,5.988,148.425
C03435=1217.234,168.435,-54.026,-177.831,5.989,148.425
C03436=1217.229,168.684,-54.048,-177.829,5.991,148.424
C03437=1217.225,168.933,-54.070,-177.826,5.992,148.424
C03438=1217.219,169.182,-54.092,-177.824,5.993,148.424
C03439=1217.215,169.431,-54.115,-177.821,5.995,148.423
C03440=1217.210,169.679,-54.137,-177.818,5.997,148.423
C03441=1217.206,169.929,-54.159,-177.816,5.998,148.422
C03442=1217.201,170.178,-54.181,-177.813,6.000,148.422
C03443=1217.196,170.427,-54.203,-177.811,6.001,148.422
C03444=1217.192,170.675,-54.226,-177.808,6.002,148.421
C03445=1217.187,170.924,-54.248,-177.805,6.004,148.421
C03446=1217.182,171.174,-54.270,-177.803,6.006,148.420
C03447=1217.178,171.423,-54.292,-177.801,6.007,148.420
C03448=1217.174,171.671,-54.315,-177.798,6.008,148.420
C03449=1217.169,171.920,-54.336,-177.795,6.010,148.419
C03450=1217.164,172.170,-54.359,-177.793,6.011,148.419
C03451=1217.159,172.418,-54.381,-177.790,6.013,148.418
C03452=1217.155,172.667,-54.403,-177.787,6.015,148.418
C03453=1217.150,172.917,-54.426,-177.785,6.015,148.417
C03454=1217.145,173.165,-54.448,-177.782,6.017,148.417
C03455=1217.141,173.414,-54.471,-177.780,6.019,148.417
C03456=1217.135,173.663,-54.493,-177.777,6.020,148.416
C03457=1217.131,173.912,-54.515,-177.775,6.022,148.416
C03458=1217.127,174.161,-54.538,-177.772,6.023,148.415
C03459=1217.122,174.410,-54.560,-177.770,6.024,148.415
C03460=1217.117,174.659,-54.582,-177.767,6.026,148.414
C03461=1217.113,174.907,-54.604,-177.764,6.028,148.414
C03462=1217.108,175.157,-54.627,-177.762,6.030,148.414
C03463=1217.104,175.406,-54.650,-177.759,6.030,148.413
C03464=1217.098,175.655,-54.672,-177.756,6.032,148.413
C03465=1217.094,175.904,-54.694,-177.754,6.034,148.412
C03466=1217.090,176.153,-54.717,-177.752,6.035,148.412
C03467=1217.084,176.402,-54.739,-177.749,6.037,148.412
C03468=1217.080,176.650,-54.762,-177.746,6.038,148.411
C03469=1217.075,176.900,-54.785,-177.743,6.040,148.411
C03470=1217.071,177.148,-54.807,-177.741,6.041,148.410
C03471=1217.066,177.398,-54.830,-177.738,6.043,148.410
C03472=1217.062,177.646,-54.852,-177.736,6.045,148.410
C03473=1217.057,177.895,-54.874,-177.734,6.046,148.409
C03474=1217.052,178.144,-54.897,-177.730,6.047,148.409
C03475=1217.048,178.393,-54.919,-177.728,6.049,148.408
C03476=1217.043,178.642,-54.942,-177.725,6.051,148.408
C03477=1217.038,178.891,-54.965,-177.723,6.052,148.408
C03478=1217.034,179.140,-54.988,-177.720,6.054,148.407
C03479=1217.029,179.388,-55.010,-177.718,6.056,148.407
C03480=1217.024,179.638,-55.033,-177.715,6.056,148.406
C03481=1217.020,179.887,-55.056,-177.713,6.058,148.406
C03482=1217.015,180.136,-55.078,-177.710,6.060,148.406
C03483=1217.011,180.384,-55.101,-177.707,6.062,148.405
C03484=1217.006,180.633,-55.124,-177.705,6.063,148.405
C03485=1217.002,180.883,-55.146,-177.702,6.064,148.404
C03486=1216.996,181.131,-55.169,-177.699,6.066,148.404
C03487=1216.992,181.380,-55.192,-177.697,6.068,148.404
C03488=1216.987,181.629,-55.215,-177.695,6.069,148.403
C03489=1216.983,181.878,-55.238,-177.692,6.071,148.403
C03490=1216.978,182.126,-55.260,-177.689,6.072,148.402
C03491=1216.973,182.376,-55.283,-177.687,6.074,148.402
C03492=1216.969,182.625,-55.306,-177.684,6.075,148.401
C03493=1216.964,182.874,-55.329,-177.681,6.077,148.401
C03494=1216.959,183.123,-55.351,-177.679,6.079,148.401
C03495=1216.955,183.371,-55.374,-177.676,6.080,148.400
C03496=1216.950,183.620,-55.397,-177.674,6.081,148.400
C03497=1216.946,183.869,-55.420,-177.671,6.083,148.400
C03498=1216.942,184.118,-55.444,-177.669,6.085,148.399
C03499=1216.936,184.367,-55.466,-177.666,6.087,148.399
C03500=1216.932,184.616,-55.489,-177.663,6.088,148.398
C03501=1216.927,184.865,-55.512,-177.661,6.089,148.398
C03502=1216.922,185.135,-55.537,-177.658,6.091,148.398
C03503=1216.917,185.404,-55.561,-177.655,6.093,148.397
C03504=1216.912,185.674,-55.586,-177.652,6.095,148.397
C03505=1216.907,185.943,-55.611,-177.650,6.096,148.396
C03506=1216.903,186.192,-55.634,-177.647,6.098,148.396
C03507=1216.898,186.441,-55.658,-177.644,6.100,148.396
C03508=1216.893,186.690,-55.681,-177.642,6.101,148.395
C03509=1216.889,186.938,-55.703,-177.639,6.103,148.395
C03510=1216.884,187.187,-55.727,-177.637,6.104,148.394
C03511=1216.879,187.437,-55.750,-177.634,6.106,148.394
C03512=1216.875,187.686,-55.772,-177.631,6.108,148.394
C03513=1216.870,187.935,-55.796,-177.629,6.109,148.393
C03514=1216.866,188.184,-55.819,-177.626,6.111,148.393
C03515=1216.861,188.433,-55.842,-177.624,6.113,148.393
C03516=1216.856,188.681,-55.865,-177.621,6.115,148.392
C03517=1216.852,188.930,-55.888,-177.619,6.116,148.392
C03518=1216.847,189.179,-55.911,-177.616,6.117,148.391
C03519=1216.842,189.428,-55.935,-177.613,6.119,148.391
C03520=1216.838,189.677,-55.958,-177.611,6.121,148.391
C03521=1216.834,189.926,-55.981,-177.608,6.123,148.390
C03522=1216.829,190.175,-56.004,-177.606,6.124,148.390
C03523=1216.824,190.424,-56.028,-177.603,6.125,148.390
C03524=1216.819,190.672,-56.051,-177.601,6.127,148.389
C03525=1216.814,190.921,-56.074,-177.598,6.129,148.389
C03526=1216.811,191.169,-56.097,-177.595,6.131,148.388
C03527=1216.806,191.418,-56.121,-177.593,6.132,148.388
C03528=1216.801,191.667,-56.144,-177.590,6.133,148.388
C03529=1216.797,191.916,-56.167,-177.587,6.135,148.387
C03530=1216.792,192.165,-56.191,-177.585,6.137,148.387
C03531=1216.787,192.415,-56.214,-177.582,6.139,148.386
C03532=1216.782,192.664,-56.238,-177.580,6.141,148.386
C03533=1216.779,192.912,-56.260,-177.577,6.142,148.386
C03534=1216.774,193.161,-56.284,-177.575,6.144,148.385
C03535=1216.769,193.410,-56.308,-177.572,6.145,148.385
C03536=1216.765,193.659,-56.331,-177.569,6.147,148.385
C03537=1216.760,193.908,-56.354,-177.567,6.149,148.384
C03538=1216.755,194.157,-56.378,-177.565,6.150,148.384
C03539=1216.750,194.405,-56.401,-177.562,6.152,148.384
C03540=1216.746,194.654,-56.425,-177.559,6.154,148.383
C03541=1216.741,194.903,-56.448,-177.556,6.155,148.383
C03542=1216.736,195.152,-56.472,-177.554,6.157,148.382
C03543=1216.732,195.401,-56.495,-177.551,6.159,148.382
C03544=1216.727,195.649,-56.519,-177.549,6.160,148.382
C03545=1216.722,195.898,-56.542,-177.546,6.162,148.381
C03546=1216.718,196.147,-56.566,-177.544,6.164,148.381
C03547=1216.713,196.396,-56.589,-177.541,6.165,148.381
C03548=1216.709,196.645,-56.613,-177.538,6.167,148.380
C03549=1216.704,196.894,-56.637,-177.536,6.169,148.380
C03550=1216.699,197.143,-56.660,-177.534,6.170,148.380
C03551=1216.695,197.391,-56.684,-177.531,6.172,148.379
C03552=1216.690,197.640,-56.707,-177.528,6.174,148.379
C03553=1216.685,197.889,-56.731,-177.526,6.176,148.379
C03554=1216.682,198.138,-56.755,-177.523,6.177,148.378
C03555=1216.677,198.387,-56.778,-177.520,6.179,148.378
C03556=1216.673,198.636,-56.803,-177.518,6.181,148.377
C03557=1216.668,198.885,-56.826,-177.516,6.182,148.377
C03558=1216.663,199.134,-56.849,-177.513,6.184,148.377
C03559=1216.659,199.382,-56.873,-177.510,6.185,148.376
C03560=1216.654,199.631,-56.897,-177.507,6.187,148.376
C03561=1216.650,199.880,-56.921,-177.505,6.189,148.376
C03562=1216.645,200.129,-56.944,-177.502,6.191,148.375
C03563=1216.641,200.377,-56.968,-177.499,6.193,148.375
C03564=1216.636,200.626,-56.992,-177.497,6.194,148.374
C03565=1216.631,200.874,-57.016,-177.495,6.196,148.374
C03566=1216.627,201.124,-57.039,-177.492,6.197,148.374
C03567=1216.622,201.372,-57.064,-177.489,6.199,148.373
C03568=1216.617,201.621,-57.087,-177.487,6.201,148.373
C03569=1216.613,201.870,-57.111,-177.484,6.203,148.373
C03570=1216.608,202.119,-57.135,-177.481,6.205,148.372
C03571=1216.604,202.368,-57.159,-177.479,6.207,148.372
C03572=1216.599,202.617,-57.182,-177.477,6.208,148.372
C03573=1216.595,202.865,-57.206,-177.474,6.210,148.371
C03574=1216.590,203.115,-57.230,-177.471,6.211,148.371
C03575=1216.585,203.363,-57.254,-177.469,6.213,148.371
C03576=1216.581,203.611,-57.278,-177.466,6.215,148.370
C03577=1216.577,203.861,-57.302,-177.463,6.217,148.370
C03578=1216.572,204.110,-57.326,-177.461,6.219,148.370
C03579=1216.567,204.359,-57.350,-177.458,6.221,148.369
C03580=1216.562,204.607,-57.374,-177.456,6.222,148.369
C03581=1216.558,204.856,-57.398,-177.453,6.223,148.369
C03582=1216.553,205.105,-57.422,-177.451,6.225,148.368
C03583=1216.550,205.354,-57.446,-177.448,6.227,148.368
C03584=1216.544,205.603,-57.471,-177.446,6.229,148.368
C03585=1216.540,205.851,-57.495,-177.443,6.231,148.367
C03586=1216.535,206.100,-57.518,-177.440,6.233,148.367
C03587=1216.531,206.348,-57.542,-177.438,6.234,148.367
C03588=1216.526,206.597,-57.567,-177.435,6.236,148.366
C03589=1216.522,206.847,-57.591,-177.432,6.238,148.366
C03590=1216.517,207.095,-57.615,-177.430,6.240,148.366
C03591=1216.512,207.344,-57.639,-177.427,6.242,148.365
C03592=1216.508,207.592,-57.664,-177.425,6.243,148.365
C03593=1216.503,207.841,-57.688,-177.422,6.245,148.365
C03594=1216.499,208.091,-57.712,-177.420,6.247,148.364
C03595=1216.494,208.339,-57.736,-177.417,6.248,148.364
C03596=1216.490,208.588,-57.760,-177.414,6.250,148.364
C03597=1216.485,208.836,-57.785,-177.412,6.252,148.363
C03598=1216.480,209.085,-57.809,-177.409,6.254,148.363
C03599=1216.476,209.335,-57.833,-177.406,6.256,148.363
C03600=1216.471,209.583,-57.857,-177.404,6.258,148.362
C03601=1216.467,209.832,-57.881,-177.401,6.259,148.362
C03602=1216.462,210.080,-57.905,-177.399,6.261,148.361
C03603=1216.458,210.330,-57.930,-177.396,6.263,148.361
C03604=1216.453,210.578,-57.954,-177.393,6.265,148.361
C03605=1216.448,210.827,-57.979,-177.391,6.266,148.360
C03606=1216.444,211.097,-58.005,-177.388,6.269,148.360
C03607=1216.439,211.368,-58.032,-177.385,6.270,148.360
C03608=1216.434,211.638,-58.058,-177.383,6.272,148.359
C03609=1216.429,211.908,-58.085,-177.380,6.274,148.359
C03610=1216.424,212.157,-58.109,-177.377,6.276,148.359
C03611=1216.420,212.406,-58.134,-177.375,6.278,148.358
C03612=1216.415,212.655,-58.158,-177.372,6.280,148.358
C03613=1216.410,212.903,-58.183,-177.370,6.282,148.358
C03614=1216.406,213.153,-58.207,-177.367,6.283,148.357
C03615=1216.401,213.401,-58.232,-177.364,6.285,148.357
C03616=1216.397,213.650,-58.256,-177.362,6.287,148.357
C03617=1216.392,213.898,-58.281,-177.359,6.289,148.356
C03618=1216.388,214.148,-58.305,-177.356,6.291,148.356
C03619=1216.383,214.396,-58.330,-177.354,6.293,148.356
C03620=1216.378,214.645,-58.354,-177.351,6.294,148.355
C03621=1216.374,214.894,-58.379,-177.348,6.296,148.355
C03622=1216.369,215.142,-58.403,-177.346,6.298,148.355
C03623=1216.365,215.391,-58.428,-177.343,6.300,148.354
C03624=1216.361,215.640,-58.453,-177.341,6.302,148.354
C03625=1216.356,215.888,-58.478,-177.338,6.304,148.354
C03626=1216.352,216.138,-58.502,-177.336,6.306,148.354
C03627=1216.347,216.386,-58.527,-177.333,6.308,148.353
C03628=1216.342,216.635,-58.551,-177.331,6.310,148.353
C03629=1216.338,216.884,-58.576,-177.328,6.311,148.353
C03630=1216.334,217.132,-58.601,-177.326,6.312,148.352
C03631=1216.329,217.381,-58.625,-177.323,6.314,148.352
C03632=1216.324,217.630,-58.650,-177.321,6.316,148.352
C03633=1216.320,217.878,-58.674,-177.318,6.318,148.351
C03634=1216.315,218.127,-58.700,-177.315,6.320,148.351
C03635=1216.310,218.376,-58.725,-177.313,6.322,148.351
C03636=1216.306,218.624,-58.749,-177.310,6.324,148.350
C03637=1216.301,218.874,-58.774,-177.307,6.325,148.350
C03638=1216.297,219.122,-58.799,-177.305,6.328,148.350
C03639=1216.293,219.371,-58.824,-177.303,6.329,148.350
C03640=1216.288,219.620,-58.848,-177.300,6.331,148.349
C03641=1216.284,219.868,-58.873,-177.297,6.333,148.349
C03642=1216.279,220.117,-58.898,-177.295,6.335,148.349
C03643=1216.274,220.366,-58.923,-177.292,6.337,148.348
C03644=1216.270,220.614,-58.948,-177.289,6.339,148.348
C03645=1216.265,220.863,-58.973,-177.287,6.341,148.348
C03646=1216.261,221.112,-58.998,-177.284,6.342,148.347
C03647=1216.257,221.360,-59.023,-177.282,6.344,148.347
C03648=1216.252,221.610,-59.048,-177.279,6.346,148.347
C03649=1216.247,221.858,-59.072,-177.277,6.348,148.347
C03650=1216.243,222.107,-59.098,-177.274,6.350,148.346
C03651=1216.238,222.355,-59.122,-177.271,6.352,148.346
C03652=1216.234,222.604,-59.148,-177.269,6.354,148.346
